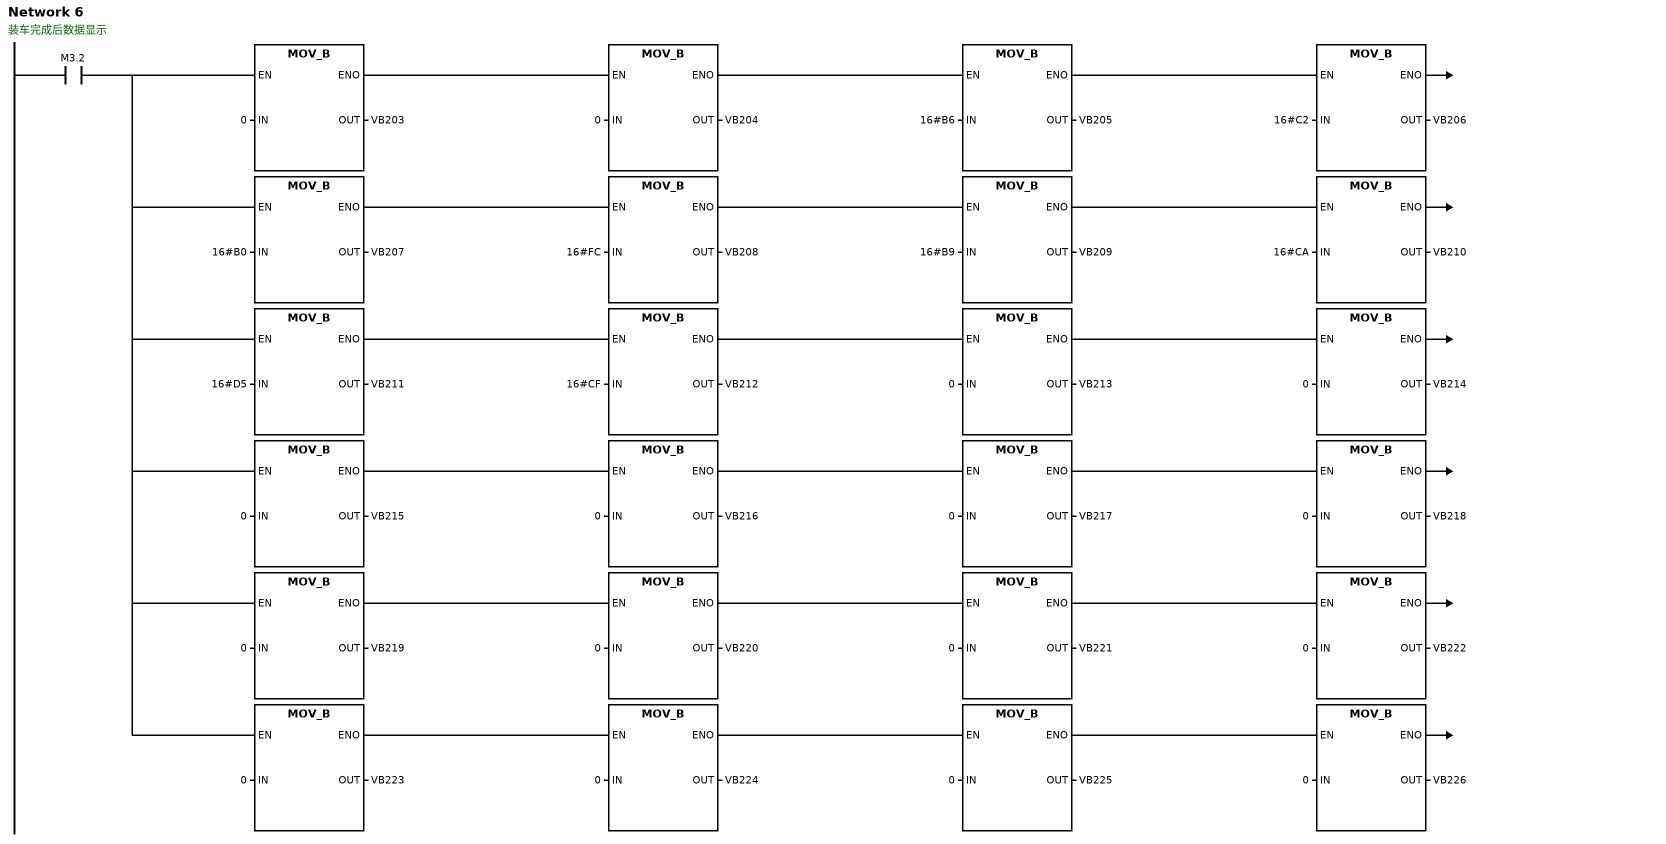
[picture p24: SBR12 networks 6-6]
Network 6
// 装车完成后数据显示
LD     M3.2
LPS
MOVB   0, VB203
AENO
MOVB   0, VB204
AENO
MOVB   16#B6, VB205
AENO
MOVB   16#C2, VB206
LRD
MOVB   16#B0, VB207
AENO
MOVB   16#FC, VB208
AENO
MOVB   16#B9, VB209
AENO
MOVB   16#CA, VB210
LRD
MOVB   16#D5, VB211
AENO
MOVB   16#CF, VB212
AENO
MOVB   0, VB213
AENO
MOVB   0, VB214
LRD
MOVB   0, VB215
AENO
MOVB   0, VB216
AENO
MOVB   0, VB217
AENO
MOVB   0, VB218
LRD
MOVB   0, VB219
AENO
MOVB   0, VB220
AENO
MOVB   0, VB221
AENO
MOVB   0, VB222
LPP
MOVB   0, VB223
AENO
MOVB   0, VB224
AENO
MOVB   0, VB225
AENO
MOVB   0, VB226
END_SUBROUTINE_BLOCK

SUBROUTINE_BLOCK LED3:SBR13
TITLE=
VAR_INPUT
D1:BYTE;	// LB0 
D2:BYTE;	// LB1 
D3:BYTE;	// LB2 
D4:BYTE;	// LB3 
P1:BYTE;	// LB4 
P2:BYTE;	// LB5 
P3:BYTE;	// LB6 
P4:BYTE;	// LB7 
P5:BYTE;	// LB8 
P6:BYTE;	// LB9 
P7:BYTE;	// LB10 
P8:BYTE;	// LB11 
RUN:WORD;	// LW12 
END_VAR
BEGIN
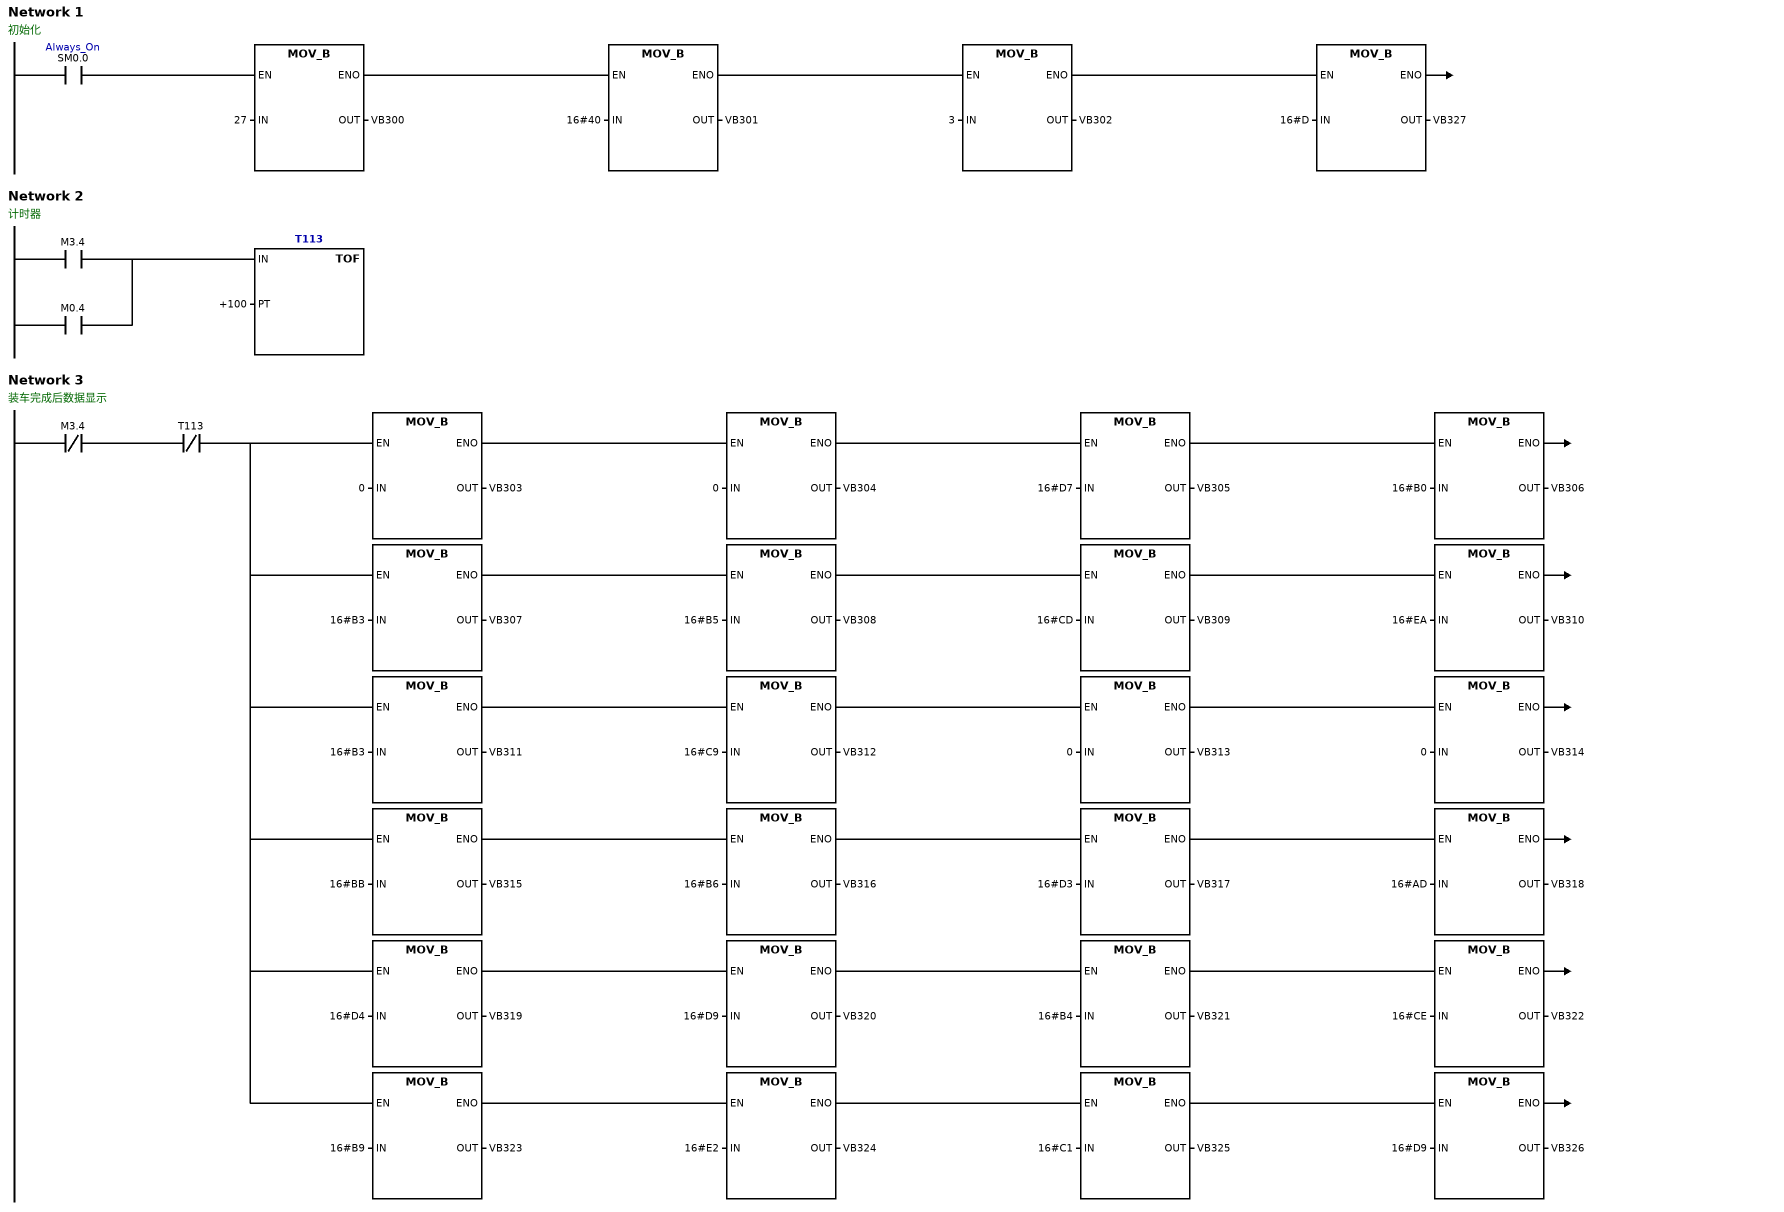
Network 1
// 初始化
LD     Always_On:SM0.0
MOVB   27, VB300
AENO
MOVB   16#40, VB301
AENO
MOVB   3, VB302
AENO
MOVB   16#D, VB327
Network 2
// 计时器
LD     M3.4
O      M0.4
TOF    T113, +100
Network 3
// 装车完成后数据显示
LDN    M3.4
AN     T113
LPS
MOVB   0, VB303
AENO
MOVB   0, VB304
AENO
MOVB   16#D7, VB305
AENO
MOVB   16#B0, VB306
LRD
MOVB   16#B3, VB307
AENO
MOVB   16#B5, VB308
AENO
MOVB   16#CD, VB309
AENO
MOVB   16#EA, VB310
LRD
MOVB   16#B3, VB311
AENO
MOVB   16#C9, VB312
AENO
MOVB   0, VB313
AENO
MOVB   0, VB314
LRD
MOVB   16#BB, VB315
AENO
MOVB   16#B6, VB316
AENO
MOVB   16#D3, VB317
AENO
MOVB   16#AD, VB318
LRD
MOVB   16#D4, VB319
AENO
MOVB   16#D9, VB320
AENO
MOVB   16#B4, VB321
AENO
MOVB   16#CE, VB322
LPP
MOVB   16#B9, VB323
AENO
MOVB   16#E2, VB324
AENO
MOVB   16#C1, VB325
AENO
MOVB   16#D9, VB326
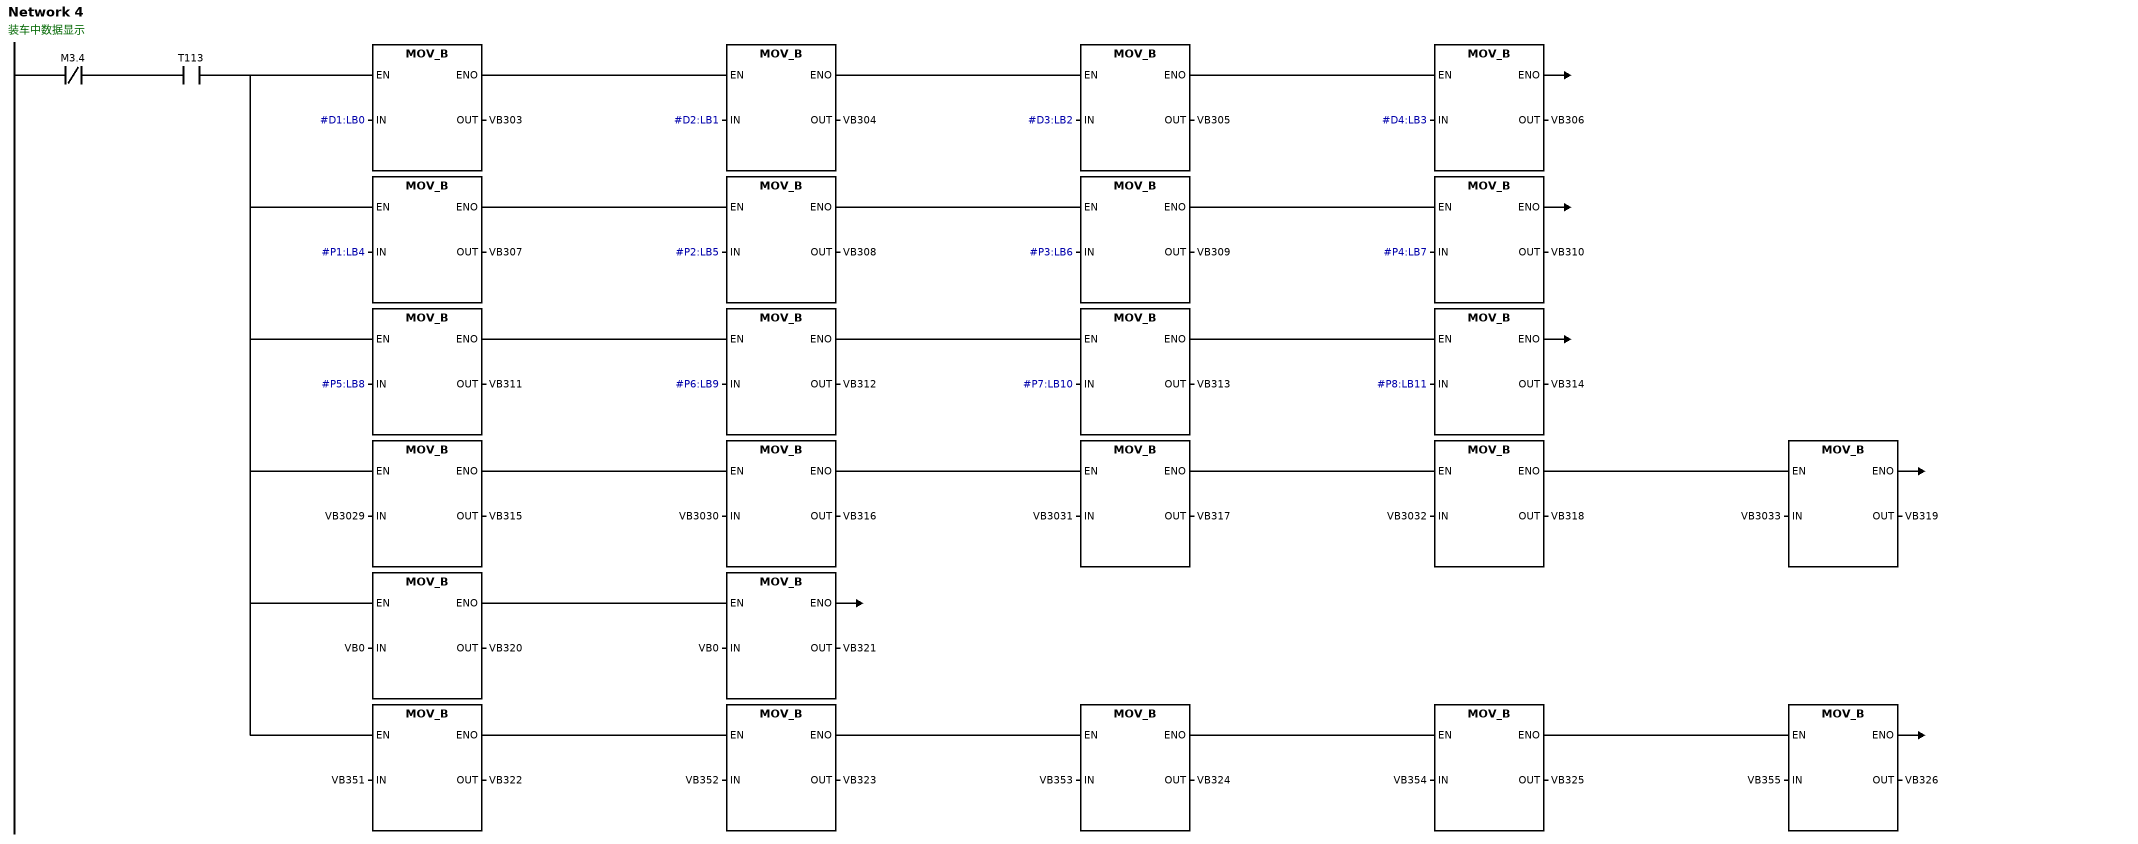
Network 4
// 装车中数据显示
LDN    M3.4
A      T113
LPS
MOVB   #D1:LB0, VB303
AENO
MOVB   #D2:LB1, VB304
AENO
MOVB   #D3:LB2, VB305
AENO
MOVB   #D4:LB3, VB306
LRD
MOVB   #P1:LB4, VB307
AENO
MOVB   #P2:LB5, VB308
AENO
MOVB   #P3:LB6, VB309
AENO
MOVB   #P4:LB7, VB310
LRD
MOVB   #P5:LB8, VB311
AENO
MOVB   #P6:LB9, VB312
AENO
MOVB   #P7:LB10, VB313
AENO
MOVB   #P8:LB11, VB314
LRD
MOVB   VB3029, VB315
AENO
MOVB   VB3030, VB316
AENO
MOVB   VB3031, VB317
AENO
MOVB   VB3032, VB318
AENO
MOVB   VB3033, VB319
LRD
MOVB   VB0, VB320
AENO
MOVB   VB0, VB321
LPP
MOVB   VB351, VB322
AENO
MOVB   VB352, VB323
AENO
MOVB   VB353, VB324
AENO
MOVB   VB354, VB325
AENO
MOVB   VB355, VB326
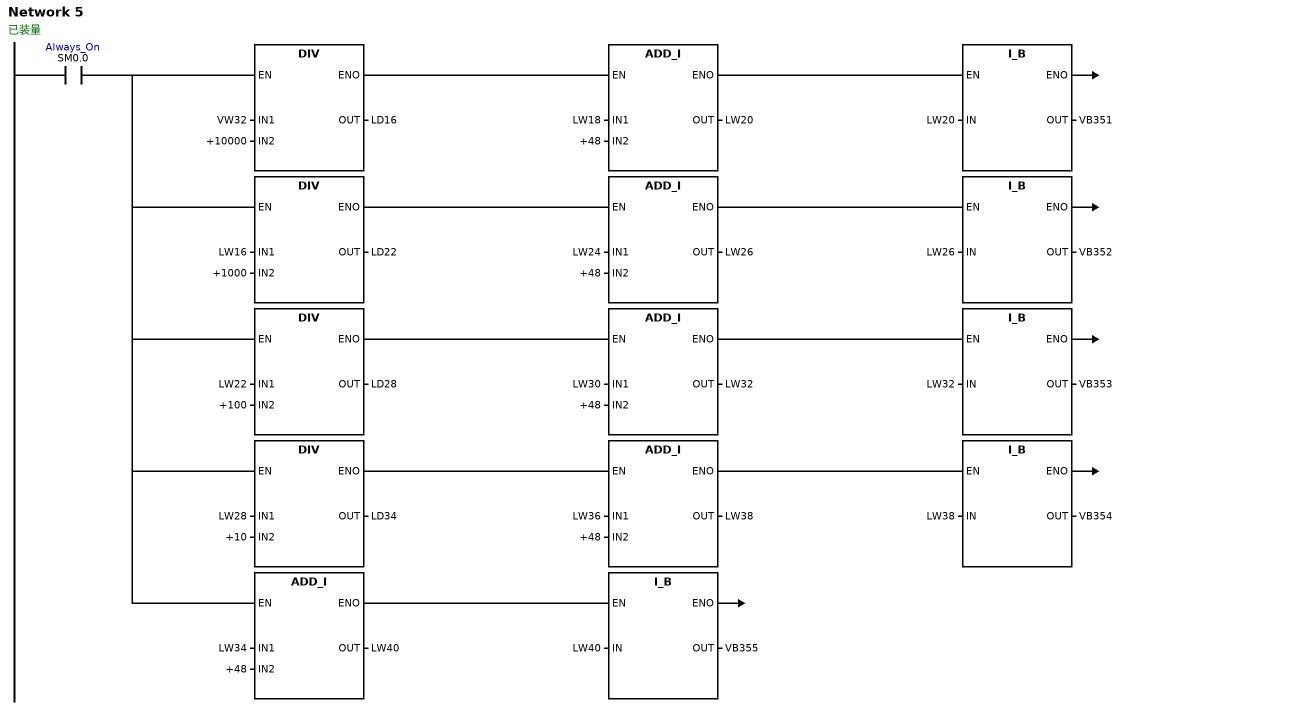
Network 5
// 已装量
LD     Always_On:SM0.0
LPS
MOVW   VW32, LW18
AENO
DIV    +10000, LD16
AENO
MOVW   LW18, LW20
AENO
+I     +48, LW20
AENO
ITB    LW20, VB351
LRD
MOVW   LW16, LW24
AENO
DIV    +1000, LD22
AENO
MOVW   LW24, LW26
AENO
+I     +48, LW26
AENO
ITB    LW26, VB352
LRD
MOVW   LW22, LW30
AENO
DIV    +100, LD28
AENO
MOVW   LW30, LW32
AENO
+I     +48, LW32
AENO
ITB    LW32, VB353
LRD
MOVW   LW28, LW36
AENO
DIV    +10, LD34
AENO
MOVW   LW36, LW38
AENO
+I     +48, LW38
AENO
ITB    LW38, VB354
LPP
MOVW   LW34, LW40
AENO
+I     +48, LW40
AENO
ITB    LW40, VB355
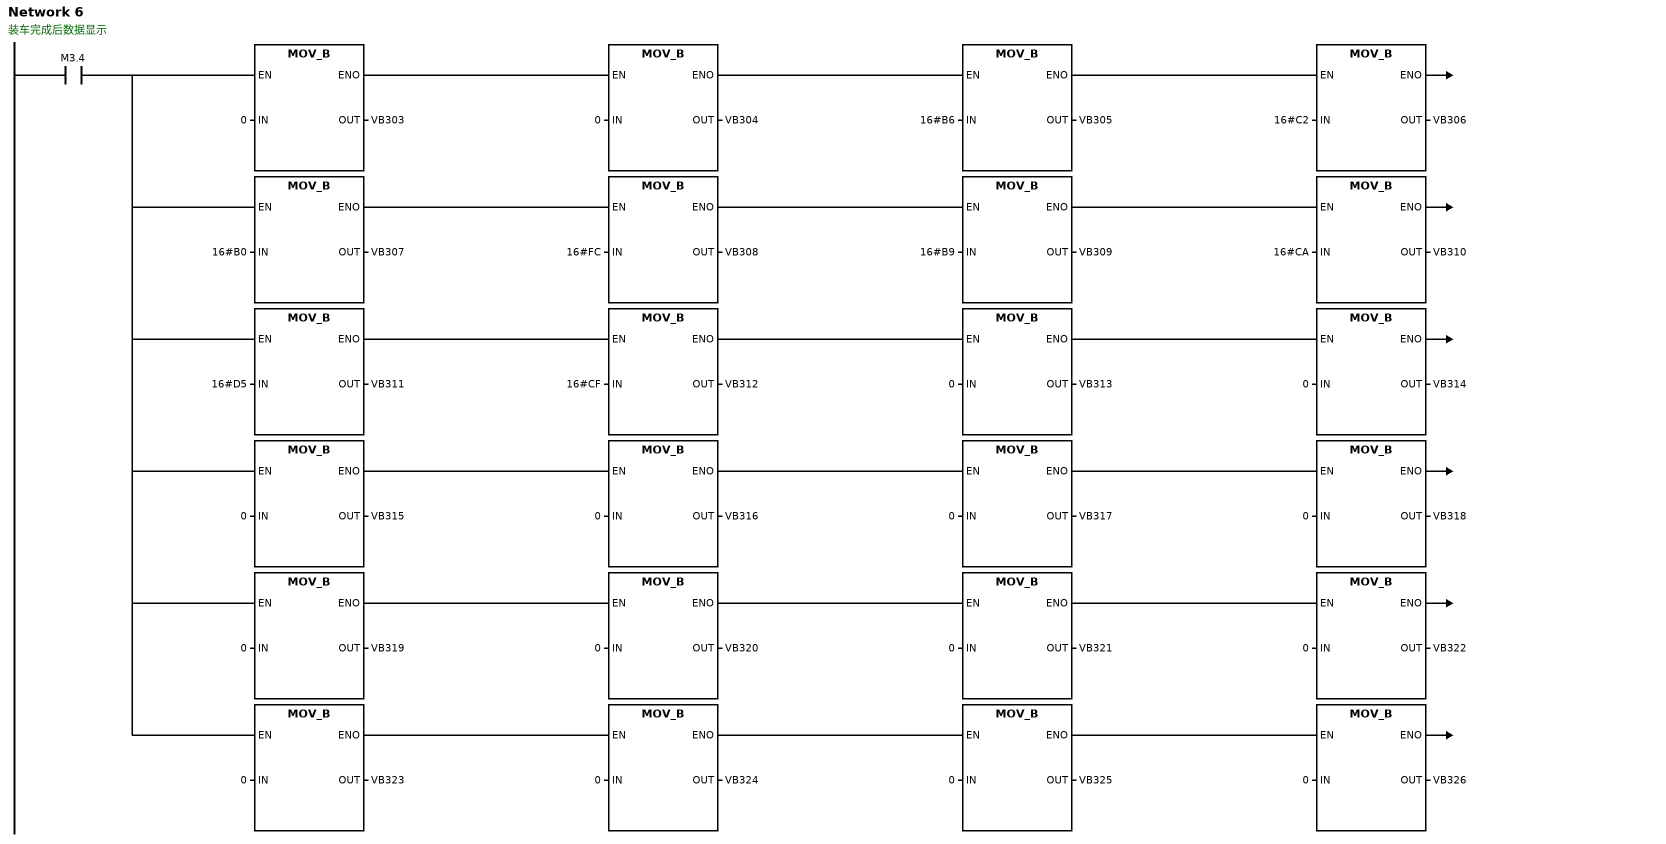
Network 6
// 装车完成后数据显示
LD     M3.4
LPS
MOVB   0, VB303
AENO
MOVB   0, VB304
AENO
MOVB   16#B6, VB305
AENO
MOVB   16#C2, VB306
LRD
MOVB   16#B0, VB307
AENO
MOVB   16#FC, VB308
AENO
MOVB   16#B9, VB309
AENO
MOVB   16#CA, VB310
LRD
MOVB   16#D5, VB311
AENO
MOVB   16#CF, VB312
AENO
MOVB   0, VB313
AENO
MOVB   0, VB314
LRD
MOVB   0, VB315
AENO
MOVB   0, VB316
AENO
MOVB   0, VB317
AENO
MOVB   0, VB318
LRD
MOVB   0, VB319
AENO
MOVB   0, VB320
AENO
MOVB   0, VB321
AENO
MOVB   0, VB322
LPP
MOVB   0, VB323
AENO
MOVB   0, VB324
AENO
MOVB   0, VB325
AENO
MOVB   0, VB326
END_SUBROUTINE_BLOCK

SUBROUTINE_BLOCK LED4:SBR14
TITLE=
VAR_INPUT
D1:BYTE;	// LB0 
D2:BYTE;	// LB1 
D3:BYTE;	// LB2 
D4:BYTE;	// LB3 
P1:BYTE;	// LB4 
P2:BYTE;	// LB5 
P3:BYTE;	// LB6 
P4:BYTE;	// LB7 
P5:BYTE;	// LB8 
P6:BYTE;	// LB9 
P7:BYTE;	// LB10 
P8:BYTE;	// LB11 
RUN:WORD;	// LW12 
END_VAR
BEGIN
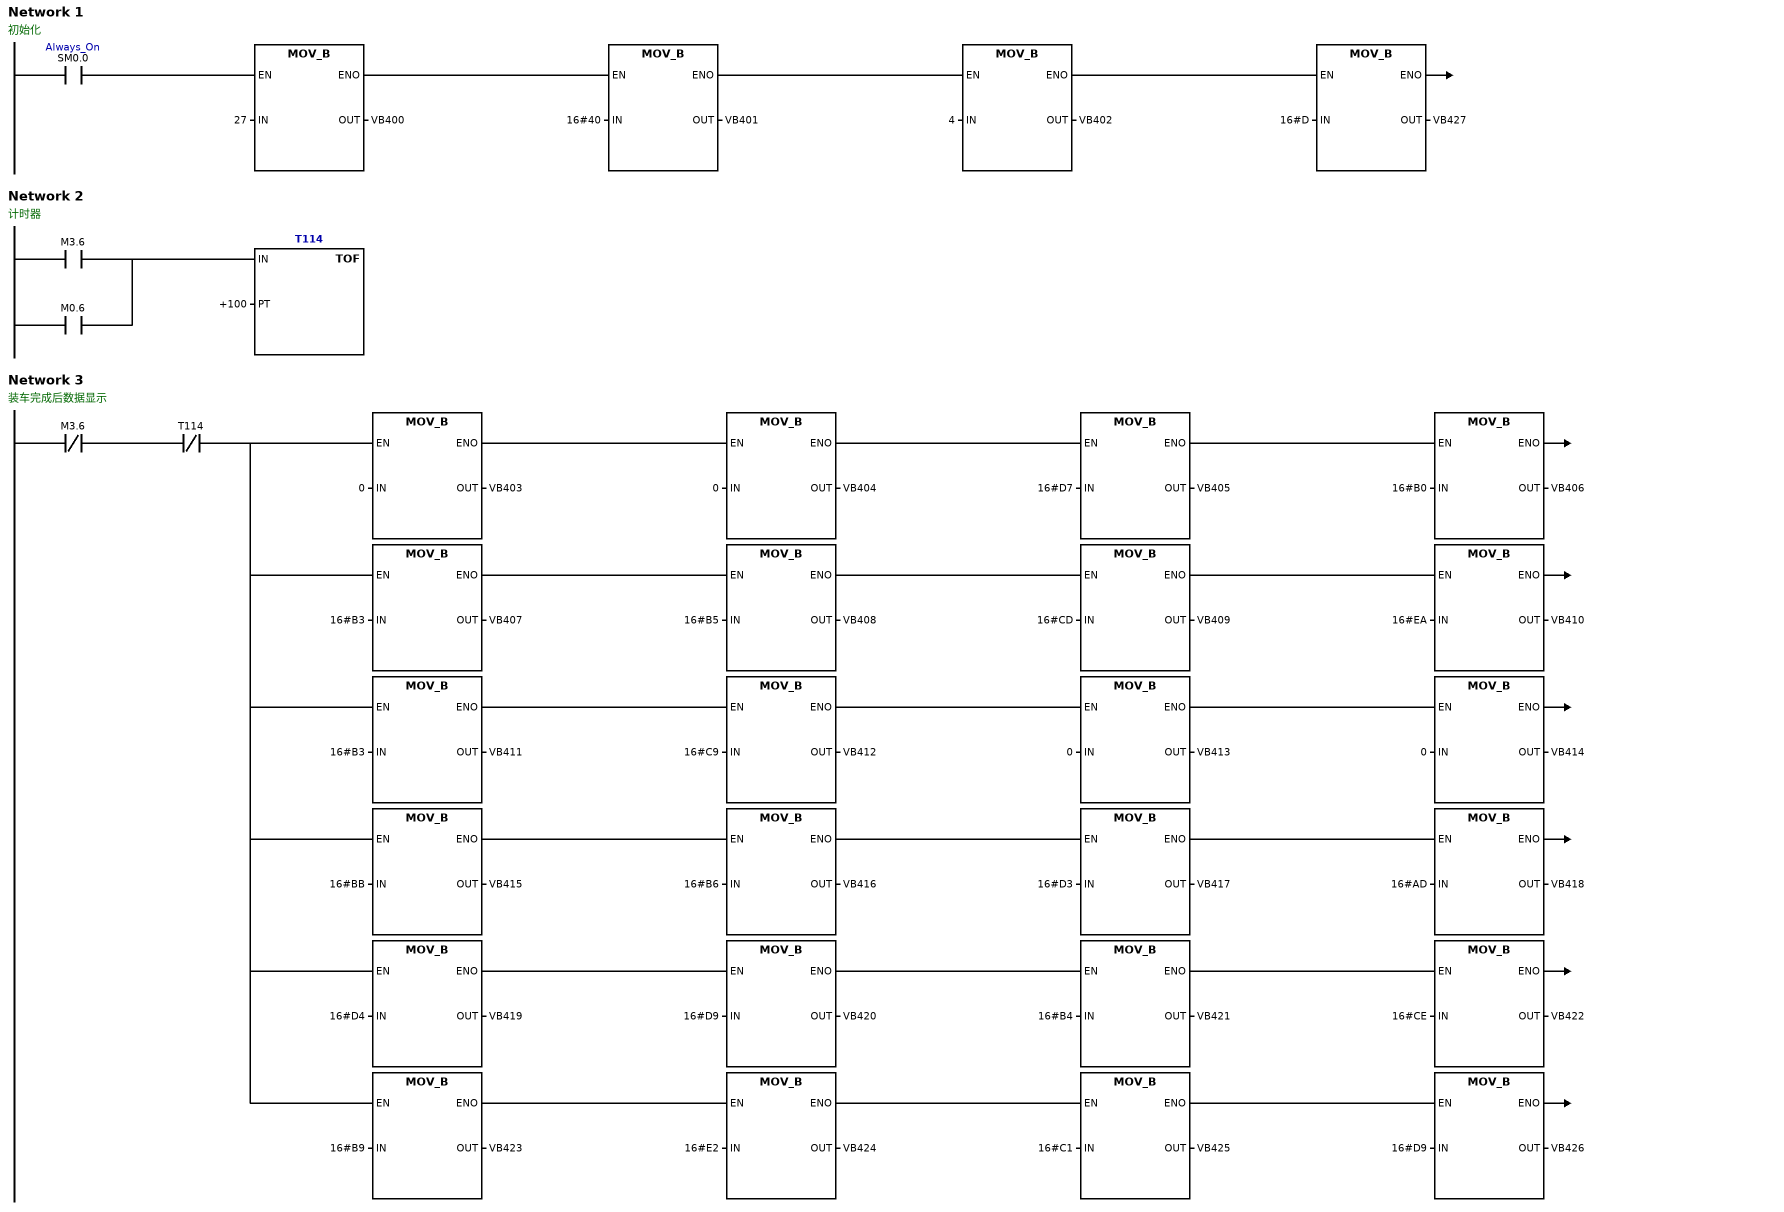
Network 1
// 初始化
LD     Always_On:SM0.0
MOVB   27, VB400
AENO
MOVB   16#40, VB401
AENO
MOVB   4, VB402
AENO
MOVB   16#D, VB427
Network 2
// 计时器
LD     M3.6
O      M0.6
TOF    T114, +100
Network 3
// 装车完成后数据显示
LDN    M3.6
AN     T114
LPS
MOVB   0, VB403
AENO
MOVB   0, VB404
AENO
MOVB   16#D7, VB405
AENO
MOVB   16#B0, VB406
LRD
MOVB   16#B3, VB407
AENO
MOVB   16#B5, VB408
AENO
MOVB   16#CD, VB409
AENO
MOVB   16#EA, VB410
LRD
MOVB   16#B3, VB411
AENO
MOVB   16#C9, VB412
AENO
MOVB   0, VB413
AENO
MOVB   0, VB414
LRD
MOVB   16#BB, VB415
AENO
MOVB   16#B6, VB416
AENO
MOVB   16#D3, VB417
AENO
MOVB   16#AD, VB418
LRD
MOVB   16#D4, VB419
AENO
MOVB   16#D9, VB420
AENO
MOVB   16#B4, VB421
AENO
MOVB   16#CE, VB422
LPP
MOVB   16#B9, VB423
AENO
MOVB   16#E2, VB424
AENO
MOVB   16#C1, VB425
AENO
MOVB   16#D9, VB426
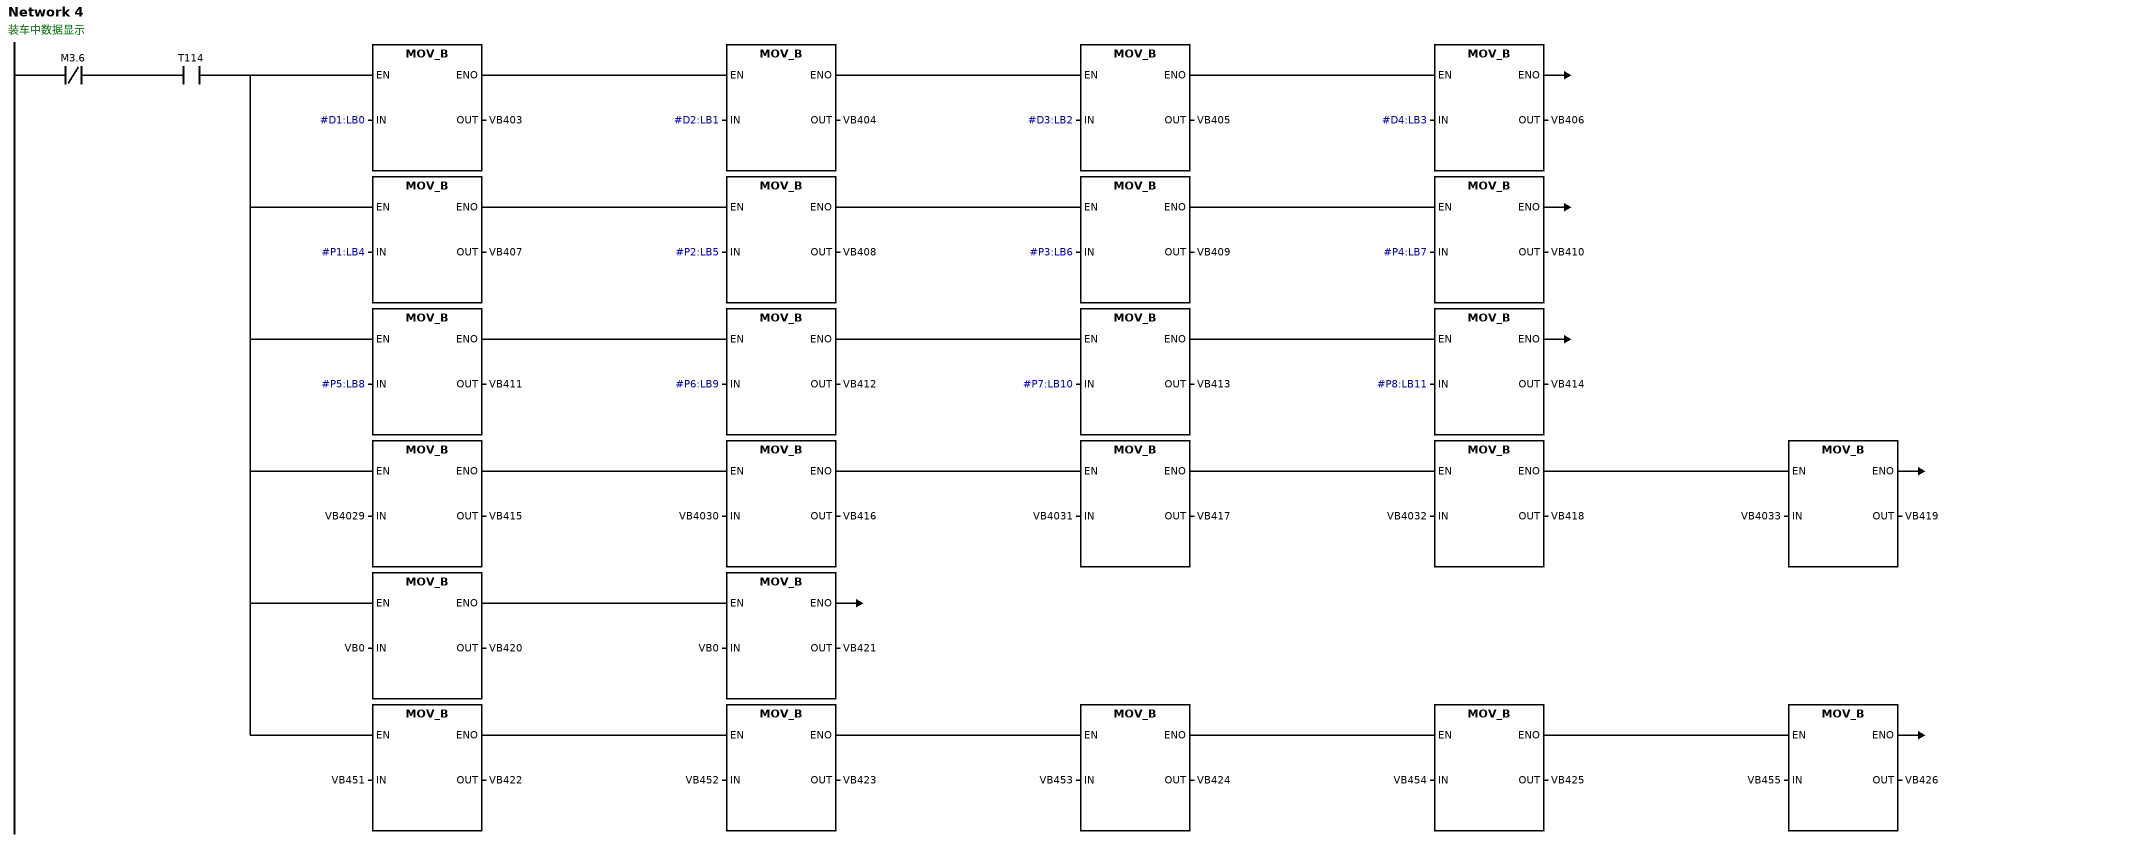
Network 4
// 装车中数据显示
LDN    M3.6
A      T114
LPS
MOVB   #D1:LB0, VB403
AENO
MOVB   #D2:LB1, VB404
AENO
MOVB   #D3:LB2, VB405
AENO
MOVB   #D4:LB3, VB406
LRD
MOVB   #P1:LB4, VB407
AENO
MOVB   #P2:LB5, VB408
AENO
MOVB   #P3:LB6, VB409
AENO
MOVB   #P4:LB7, VB410
LRD
MOVB   #P5:LB8, VB411
AENO
MOVB   #P6:LB9, VB412
AENO
MOVB   #P7:LB10, VB413
AENO
MOVB   #P8:LB11, VB414
LRD
MOVB   VB4029, VB415
AENO
MOVB   VB4030, VB416
AENO
MOVB   VB4031, VB417
AENO
MOVB   VB4032, VB418
AENO
MOVB   VB4033, VB419
LRD
MOVB   VB0, VB420
AENO
MOVB   VB0, VB421
LPP
MOVB   VB451, VB422
AENO
MOVB   VB452, VB423
AENO
MOVB   VB453, VB424
AENO
MOVB   VB454, VB425
AENO
MOVB   VB455, VB426
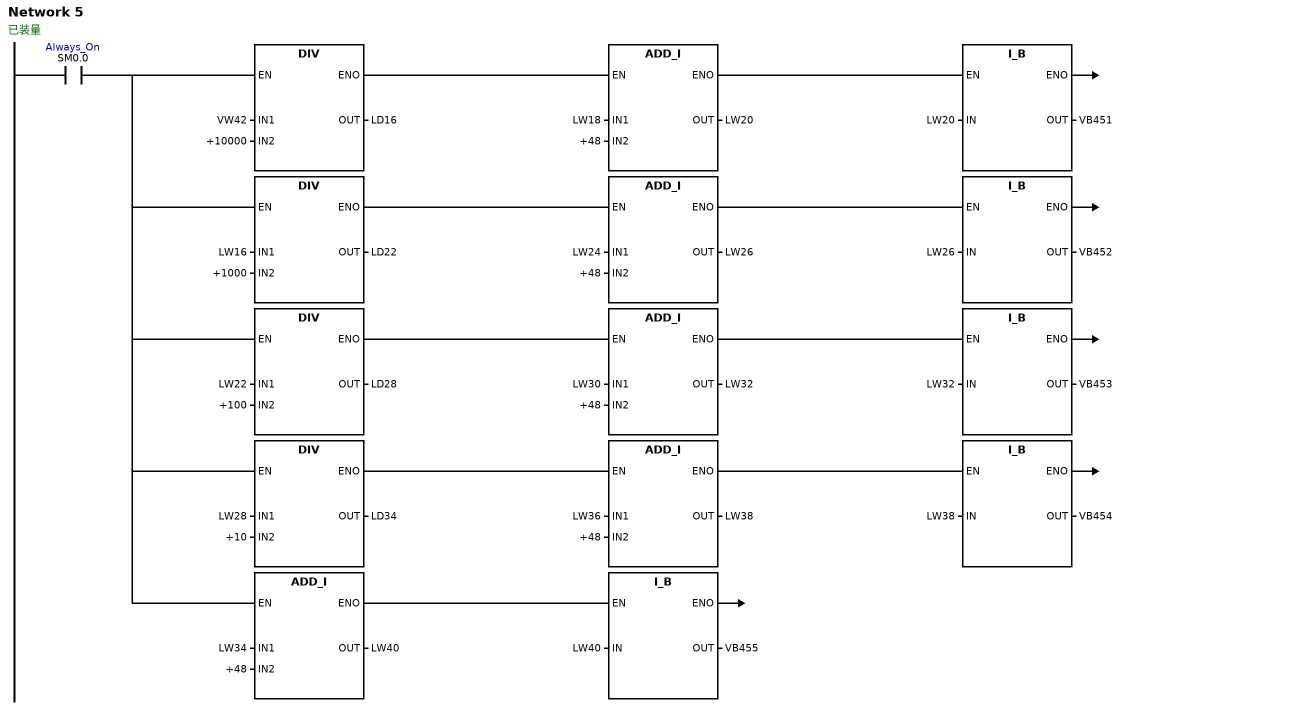
Network 5
// 已装量
LD     Always_On:SM0.0
LPS
MOVW   VW42, LW18
AENO
DIV    +10000, LD16
AENO
MOVW   LW18, LW20
AENO
+I     +48, LW20
AENO
ITB    LW20, VB451
LRD
MOVW   LW16, LW24
AENO
DIV    +1000, LD22
AENO
MOVW   LW24, LW26
AENO
+I     +48, LW26
AENO
ITB    LW26, VB452
LRD
MOVW   LW22, LW30
AENO
DIV    +100, LD28
AENO
MOVW   LW30, LW32
AENO
+I     +48, LW32
AENO
ITB    LW32, VB453
LRD
MOVW   LW28, LW36
AENO
DIV    +10, LD34
AENO
MOVW   LW36, LW38
AENO
+I     +48, LW38
AENO
ITB    LW38, VB454
LPP
MOVW   LW34, LW40
AENO
+I     +48, LW40
AENO
ITB    LW40, VB455
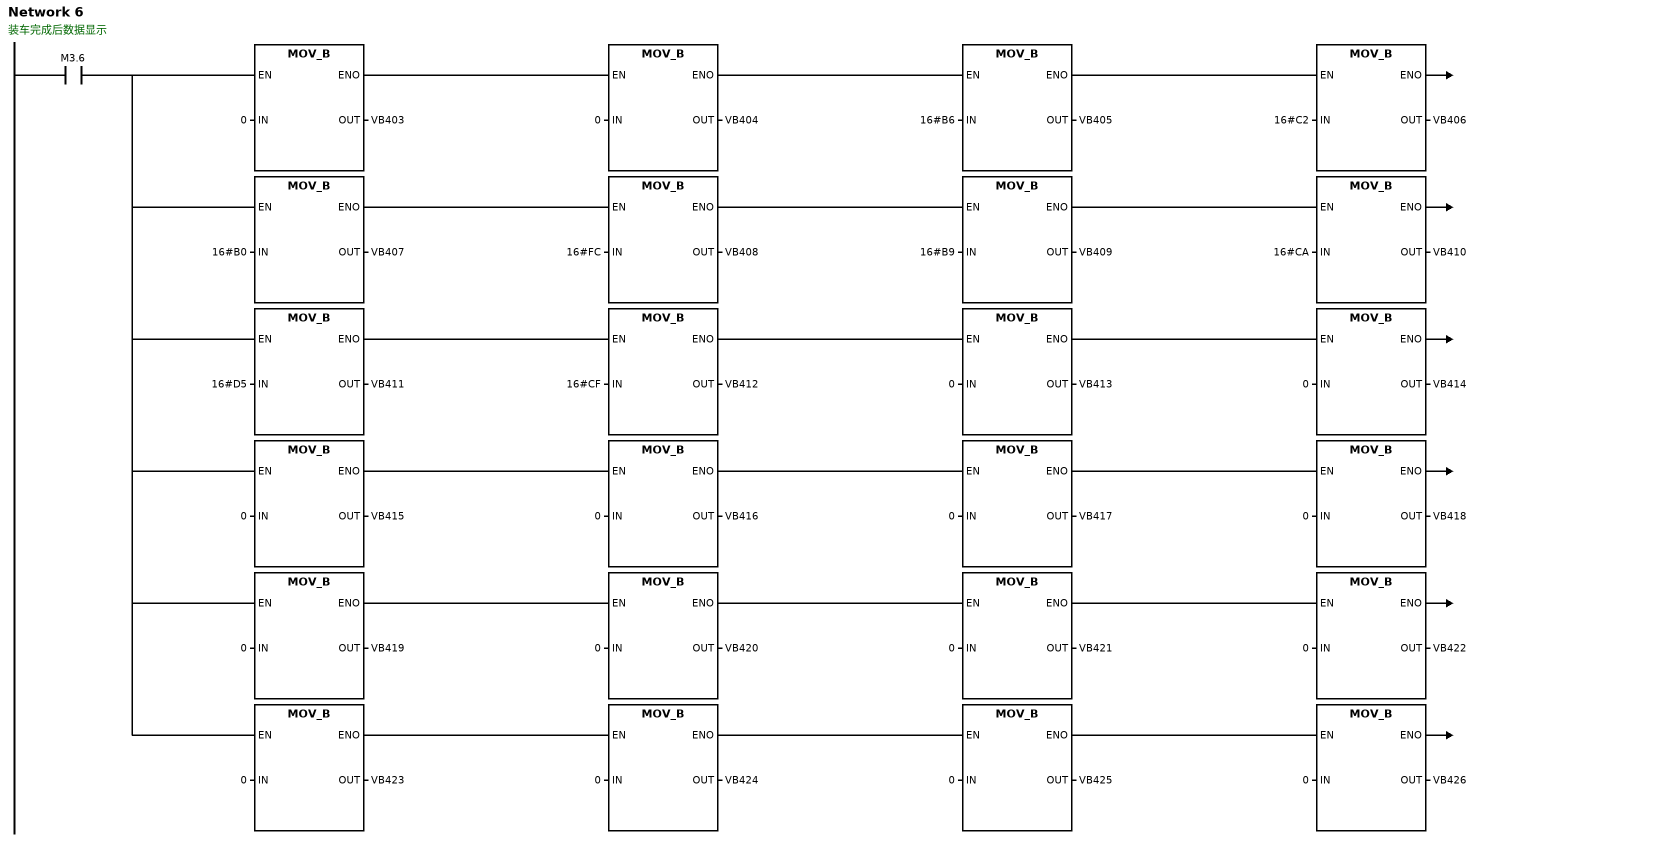
Network 6
// 装车完成后数据显示
LD     M3.6
LPS
MOVB   0, VB403
AENO
MOVB   0, VB404
AENO
MOVB   16#B6, VB405
AENO
MOVB   16#C2, VB406
LRD
MOVB   16#B0, VB407
AENO
MOVB   16#FC, VB408
AENO
MOVB   16#B9, VB409
AENO
MOVB   16#CA, VB410
LRD
MOVB   16#D5, VB411
AENO
MOVB   16#CF, VB412
AENO
MOVB   0, VB413
AENO
MOVB   0, VB414
LRD
MOVB   0, VB415
AENO
MOVB   0, VB416
AENO
MOVB   0, VB417
AENO
MOVB   0, VB418
LRD
MOVB   0, VB419
AENO
MOVB   0, VB420
AENO
MOVB   0, VB421
AENO
MOVB   0, VB422
LPP
MOVB   0, VB423
AENO
MOVB   0, VB424
AENO
MOVB   0, VB425
AENO
MOVB   0, VB426
END_SUBROUTINE_BLOCK

SUBROUTINE_BLOCK N1收:SBR21
TITLE=
VAR_OUTPUT
总袋数1:WORD;	// LW0 
袋长1:WORD;	// LW2 
END_VAR
VAR
TEMP1:WORD;	// LW4 
TEMP2:WORD;	// LW6 
TEMP3:WORD;	// LW8 
TEMP4:WORD;	// LW10 
TEMP5:WORD;	// LW12 
TEMP6:WORD;	// LW14 
TEMP7:WORD;	// LW16 
TEMP8:WORD;	// LW18 
TEMP9:WORD;	// LW20 
TEMP10:WORD;	// LW22 
TEMP11:WORD;	// LW24 
TEMP12:WORD;	// LW26 
TEMP13:WORD;	// LW28 
TEMP14:WORD;	// LW30 
TEMP15:WORD;	// LW32 
TEMP16:WORD;	// LW34 
TEMP17:WORD;	// LW36 
TEMP18:WORD;	// LW38 
TEMP19:WORD;	// LW40 
TEMP20:WORD;	// LW42 
TEMP21:WORD;	// LW44 
END_VAR
BEGIN
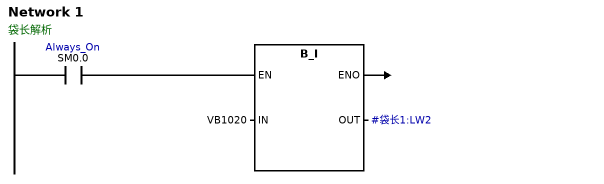
Network 1
// 袋长解析
LD     Always_On:SM0.0
BTI    VB1020, #袋长1:LW2
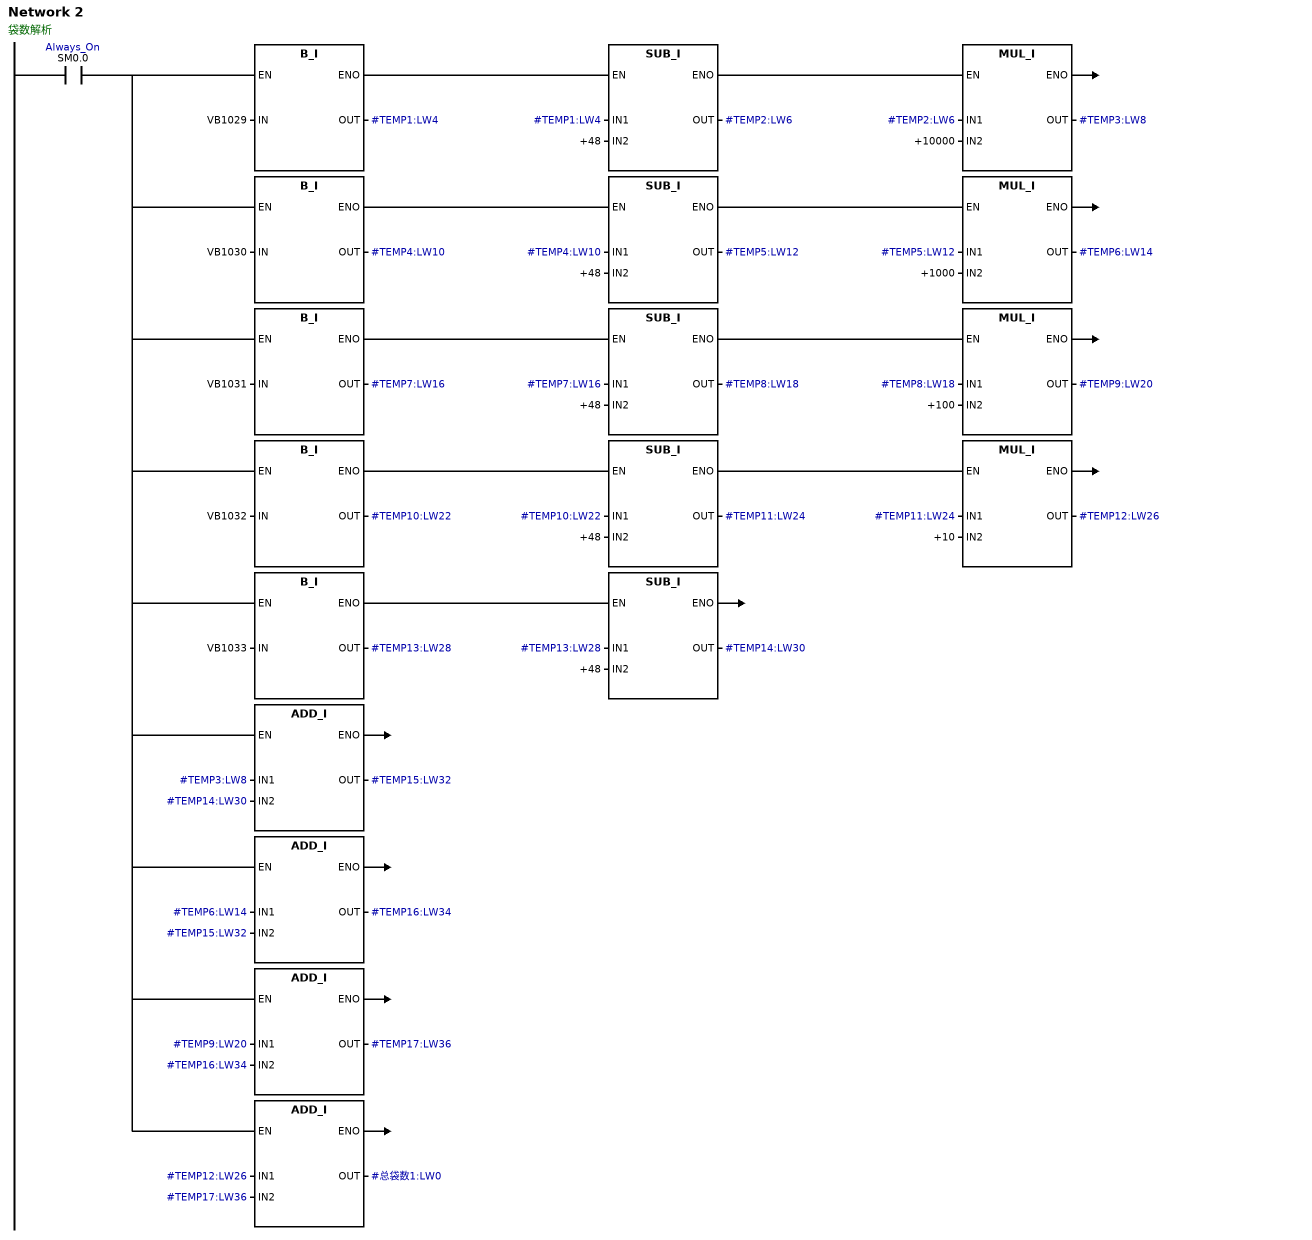
Network 2
// 袋数解析
LD     Always_On:SM0.0
LPS
BTI    VB1029, #TEMP1:LW4
AENO
MOVW   #TEMP1:LW4, #TEMP2:LW6
AENO
-I     +48, #TEMP2:LW6
AENO
MOVW   #TEMP2:LW6, #TEMP3:LW8
*I     +10000, #TEMP3:LW8
LRD
BTI    VB1030, #TEMP4:LW10
AENO
MOVW   #TEMP4:LW10, #TEMP5:LW12
AENO
-I     +48, #TEMP5:LW12
AENO
MOVW   #TEMP5:LW12, #TEMP6:LW14
*I     +1000, #TEMP6:LW14
LRD
BTI    VB1031, #TEMP7:LW16
AENO
MOVW   #TEMP7:LW16, #TEMP8:LW18
AENO
-I     +48, #TEMP8:LW18
AENO
MOVW   #TEMP8:LW18, #TEMP9:LW20
*I     +100, #TEMP9:LW20
LRD
BTI    VB1032, #TEMP10:LW22
AENO
MOVW   #TEMP10:LW22, #TEMP11:LW24
AENO
-I     +48, #TEMP11:LW24
AENO
MOVW   #TEMP11:LW24, #TEMP12:LW26
*I     +10, #TEMP12:LW26
LRD
BTI    VB1033, #TEMP13:LW28
AENO
MOVW   #TEMP13:LW28, #TEMP14:LW30
-I     +48, #TEMP14:LW30
LRD
MOVW   #TEMP3:LW8, #TEMP15:LW32
+I     #TEMP14:LW30, #TEMP15:LW32
LRD
MOVW   #TEMP6:LW14, #TEMP16:LW34
+I     #TEMP15:LW32, #TEMP16:LW34
LRD
MOVW   #TEMP9:LW20, #TEMP17:LW36
+I     #TEMP16:LW34, #TEMP17:LW36
LPP
MOVW   #TEMP12:LW26, #总袋数1:LW0
+I     #TEMP17:LW36, #总袋数1:LW0
END_SUBROUTINE_BLOCK

SUBROUTINE_BLOCK N2收:SBR22
TITLE=
VAR_OUTPUT
总袋数1:WORD;	// LW0 
袋长1:WORD;	// LW2 
END_VAR
VAR
TEMP1:WORD;	// LW4 
TEMP2:WORD;	// LW6 
TEMP3:WORD;	// LW8 
TEMP4:WORD;	// LW10 
TEMP5:WORD;	// LW12 
TEMP6:WORD;	// LW14 
TEMP7:WORD;	// LW16 
TEMP8:WORD;	// LW18 
TEMP9:WORD;	// LW20 
TEMP10:WORD;	// LW22 
TEMP11:WORD;	// LW24 
TEMP12:WORD;	// LW26 
TEMP13:WORD;	// LW28 
TEMP14:WORD;	// LW30 
TEMP15:WORD;	// LW32 
TEMP16:WORD;	// LW34 
TEMP17:WORD;	// LW36 
TEMP18:WORD;	// LW38 
TEMP19:WORD;	// LW40 
TEMP20:WORD;	// LW42 
TEMP21:WORD;	// LW44 
END_VAR
BEGIN
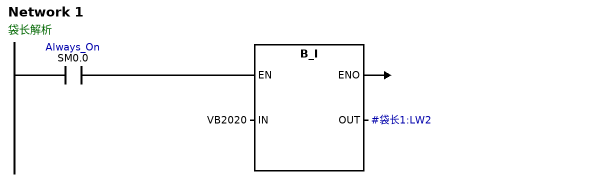
Network 1
// 袋长解析
LD     Always_On:SM0.0
BTI    VB2020, #袋长1:LW2
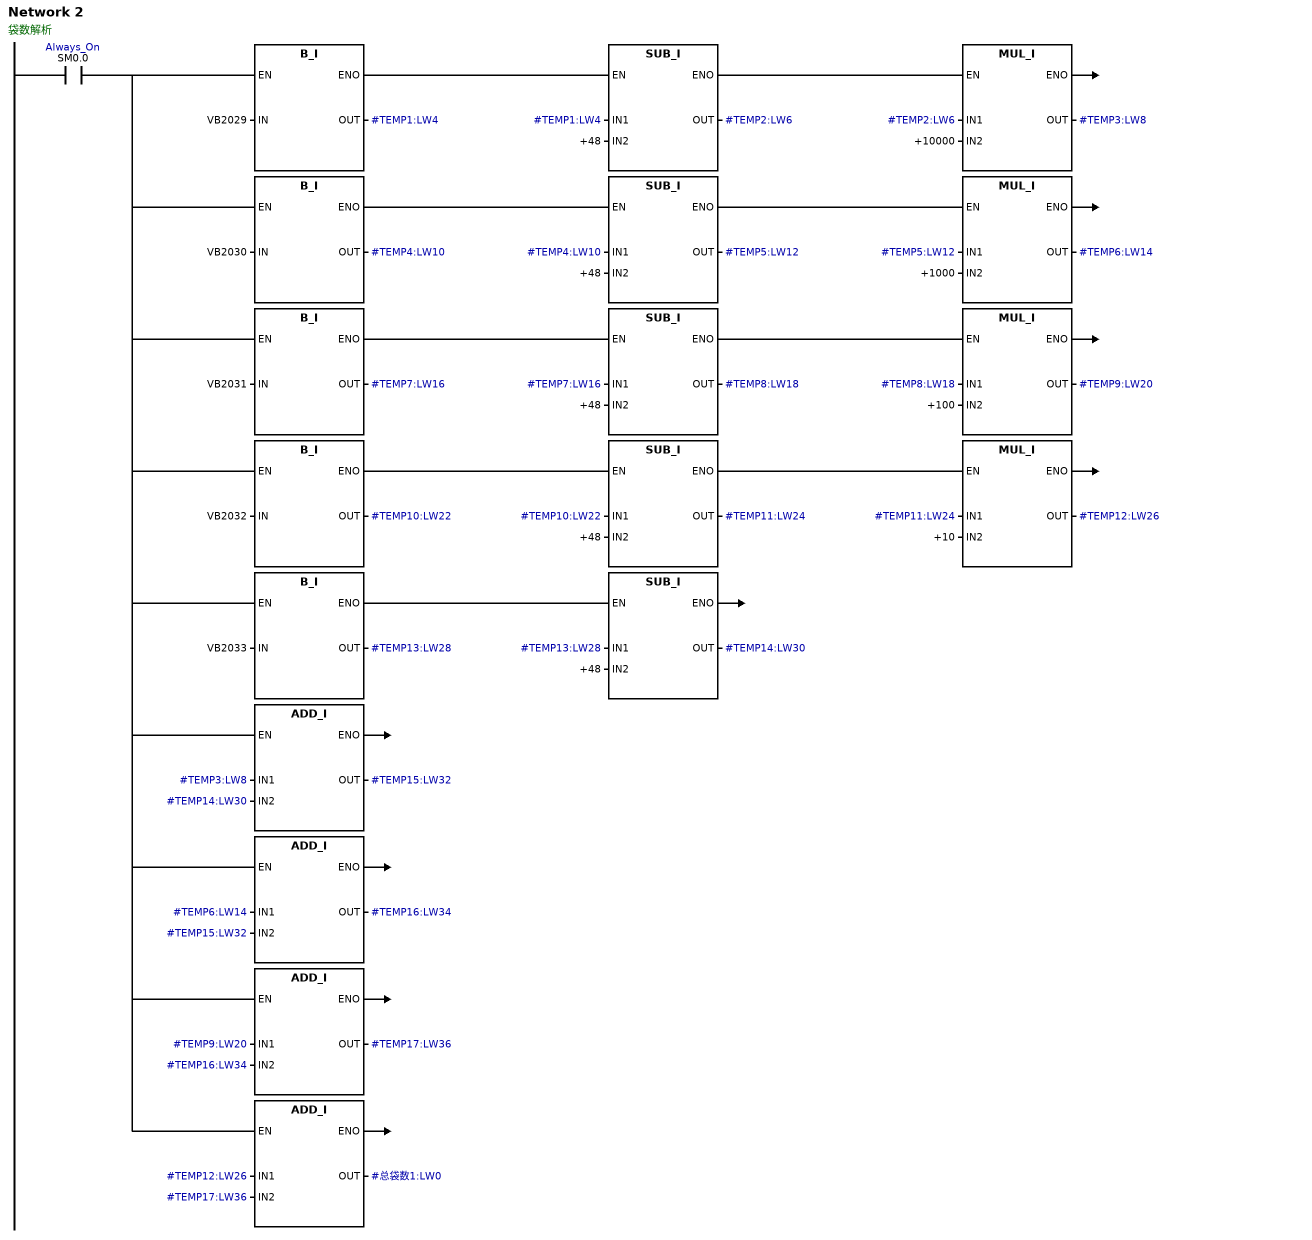
Network 2
// 袋数解析
LD     Always_On:SM0.0
LPS
BTI    VB2029, #TEMP1:LW4
AENO
MOVW   #TEMP1:LW4, #TEMP2:LW6
AENO
-I     +48, #TEMP2:LW6
AENO
MOVW   #TEMP2:LW6, #TEMP3:LW8
*I     +10000, #TEMP3:LW8
LRD
BTI    VB2030, #TEMP4:LW10
AENO
MOVW   #TEMP4:LW10, #TEMP5:LW12
AENO
-I     +48, #TEMP5:LW12
AENO
MOVW   #TEMP5:LW12, #TEMP6:LW14
*I     +1000, #TEMP6:LW14
LRD
BTI    VB2031, #TEMP7:LW16
AENO
MOVW   #TEMP7:LW16, #TEMP8:LW18
AENO
-I     +48, #TEMP8:LW18
AENO
MOVW   #TEMP8:LW18, #TEMP9:LW20
*I     +100, #TEMP9:LW20
LRD
BTI    VB2032, #TEMP10:LW22
AENO
MOVW   #TEMP10:LW22, #TEMP11:LW24
AENO
-I     +48, #TEMP11:LW24
AENO
MOVW   #TEMP11:LW24, #TEMP12:LW26
*I     +10, #TEMP12:LW26
LRD
BTI    VB2033, #TEMP13:LW28
AENO
MOVW   #TEMP13:LW28, #TEMP14:LW30
-I     +48, #TEMP14:LW30
LRD
MOVW   #TEMP3:LW8, #TEMP15:LW32
+I     #TEMP14:LW30, #TEMP15:LW32
LRD
MOVW   #TEMP6:LW14, #TEMP16:LW34
+I     #TEMP15:LW32, #TEMP16:LW34
LRD
MOVW   #TEMP9:LW20, #TEMP17:LW36
+I     #TEMP16:LW34, #TEMP17:LW36
LPP
MOVW   #TEMP12:LW26, #总袋数1:LW0
+I     #TEMP17:LW36, #总袋数1:LW0
END_SUBROUTINE_BLOCK

SUBROUTINE_BLOCK N3收:SBR23
TITLE=
VAR_OUTPUT
总袋数1:WORD;	// LW0 
袋长1:WORD;	// LW2 
END_VAR
VAR
TEMP1:WORD;	// LW4 
TEMP2:WORD;	// LW6 
TEMP3:WORD;	// LW8 
TEMP4:WORD;	// LW10 
TEMP5:WORD;	// LW12 
TEMP6:WORD;	// LW14 
TEMP7:WORD;	// LW16 
TEMP8:WORD;	// LW18 
TEMP9:WORD;	// LW20 
TEMP10:WORD;	// LW22 
TEMP11:WORD;	// LW24 
TEMP12:WORD;	// LW26 
TEMP13:WORD;	// LW28 
TEMP14:WORD;	// LW30 
TEMP15:WORD;	// LW32 
TEMP16:WORD;	// LW34 
TEMP17:WORD;	// LW36 
TEMP18:WORD;	// LW38 
TEMP19:WORD;	// LW40 
TEMP20:WORD;	// LW42 
TEMP21:WORD;	// LW44 
END_VAR
BEGIN
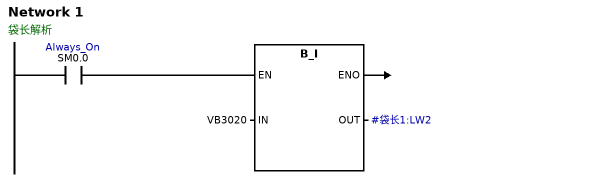
Network 1
// 袋长解析
LD     Always_On:SM0.0
BTI    VB3020, #袋长1:LW2
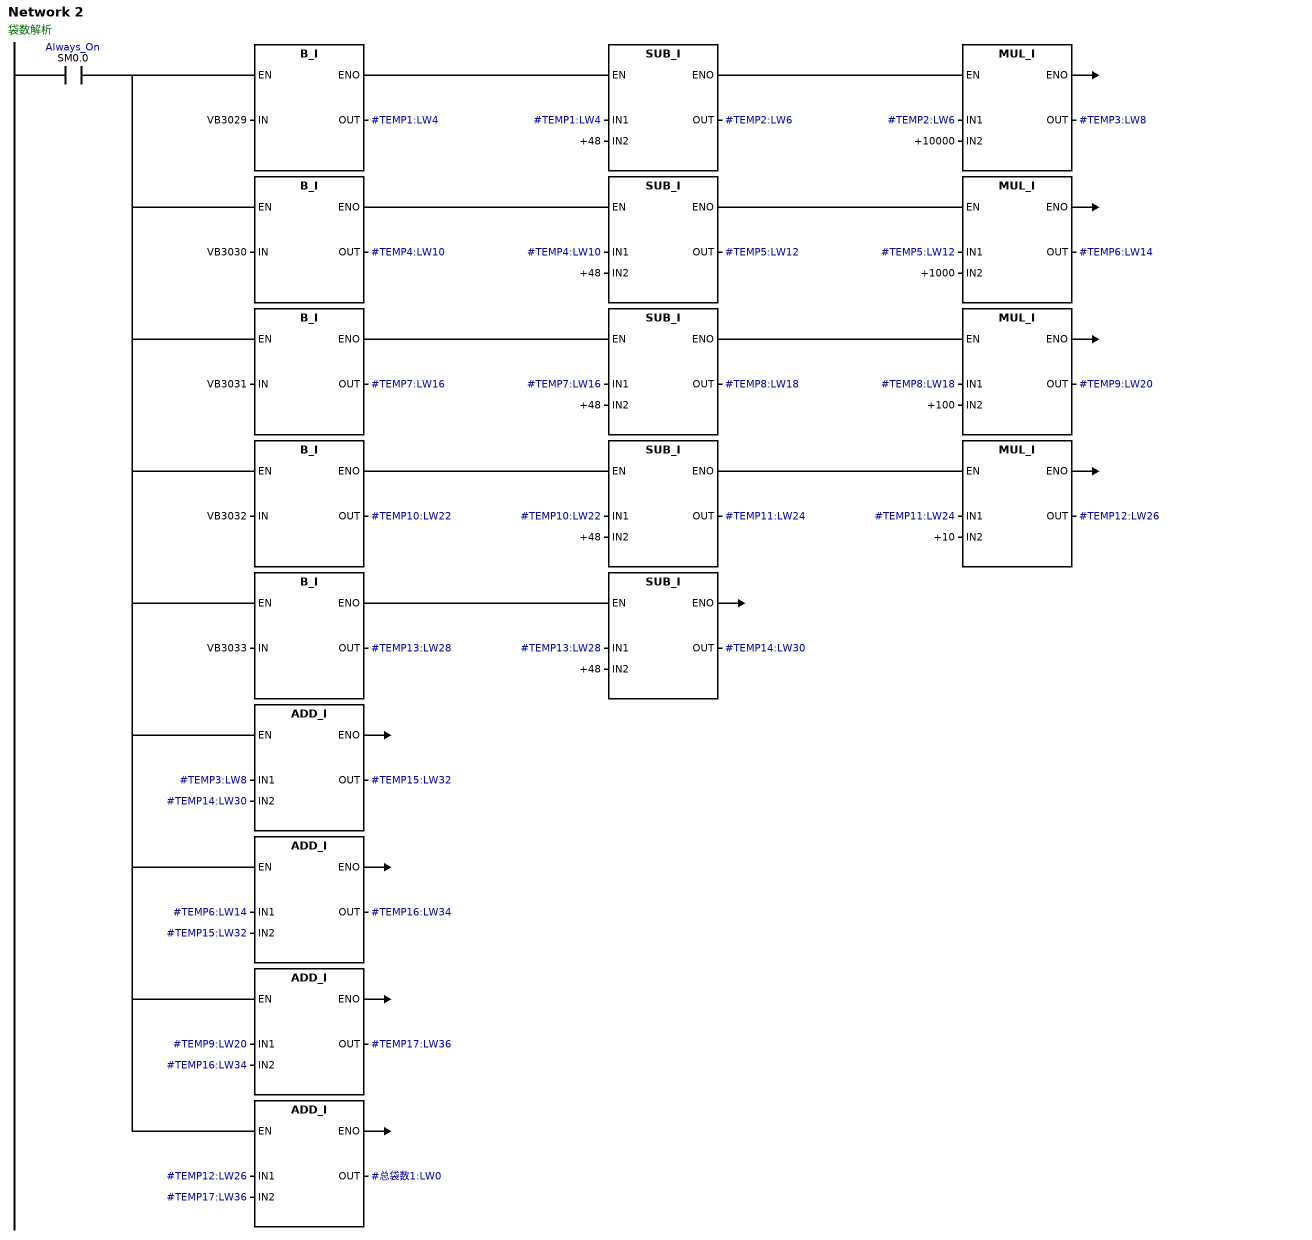
Network 2
// 袋数解析
LD     Always_On:SM0.0
LPS
BTI    VB3029, #TEMP1:LW4
AENO
MOVW   #TEMP1:LW4, #TEMP2:LW6
AENO
-I     +48, #TEMP2:LW6
AENO
MOVW   #TEMP2:LW6, #TEMP3:LW8
*I     +10000, #TEMP3:LW8
LRD
BTI    VB3030, #TEMP4:LW10
AENO
MOVW   #TEMP4:LW10, #TEMP5:LW12
AENO
-I     +48, #TEMP5:LW12
AENO
MOVW   #TEMP5:LW12, #TEMP6:LW14
*I     +1000, #TEMP6:LW14
LRD
BTI    VB3031, #TEMP7:LW16
AENO
MOVW   #TEMP7:LW16, #TEMP8:LW18
AENO
-I     +48, #TEMP8:LW18
AENO
MOVW   #TEMP8:LW18, #TEMP9:LW20
*I     +100, #TEMP9:LW20
LRD
BTI    VB3032, #TEMP10:LW22
AENO
MOVW   #TEMP10:LW22, #TEMP11:LW24
AENO
-I     +48, #TEMP11:LW24
AENO
MOVW   #TEMP11:LW24, #TEMP12:LW26
*I     +10, #TEMP12:LW26
LRD
BTI    VB3033, #TEMP13:LW28
AENO
MOVW   #TEMP13:LW28, #TEMP14:LW30
-I     +48, #TEMP14:LW30
LRD
MOVW   #TEMP3:LW8, #TEMP15:LW32
+I     #TEMP14:LW30, #TEMP15:LW32
LRD
MOVW   #TEMP6:LW14, #TEMP16:LW34
+I     #TEMP15:LW32, #TEMP16:LW34
LRD
MOVW   #TEMP9:LW20, #TEMP17:LW36
+I     #TEMP16:LW34, #TEMP17:LW36
LPP
MOVW   #TEMP12:LW26, #总袋数1:LW0
+I     #TEMP17:LW36, #总袋数1:LW0
END_SUBROUTINE_BLOCK

SUBROUTINE_BLOCK N4收:SBR24
TITLE=
VAR_OUTPUT
总袋数1:WORD;	// LW0 
袋长1:WORD;	// LW2 
END_VAR
VAR
TEMP1:WORD;	// LW4 
TEMP2:WORD;	// LW6 
TEMP3:WORD;	// LW8 
TEMP4:WORD;	// LW10 
TEMP5:WORD;	// LW12 
TEMP6:WORD;	// LW14 
TEMP7:WORD;	// LW16 
TEMP8:WORD;	// LW18 
TEMP9:WORD;	// LW20 
TEMP10:WORD;	// LW22 
TEMP11:WORD;	// LW24 
TEMP12:WORD;	// LW26 
TEMP13:WORD;	// LW28 
TEMP14:WORD;	// LW30 
TEMP15:WORD;	// LW32 
TEMP16:WORD;	// LW34 
TEMP17:WORD;	// LW36 
TEMP18:WORD;	// LW38 
TEMP19:WORD;	// LW40 
TEMP20:WORD;	// LW42 
TEMP21:WORD;	// LW44 
END_VAR
BEGIN
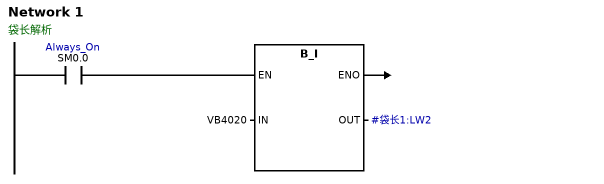
Network 1
// 袋长解析
LD     Always_On:SM0.0
BTI    VB4020, #袋长1:LW2
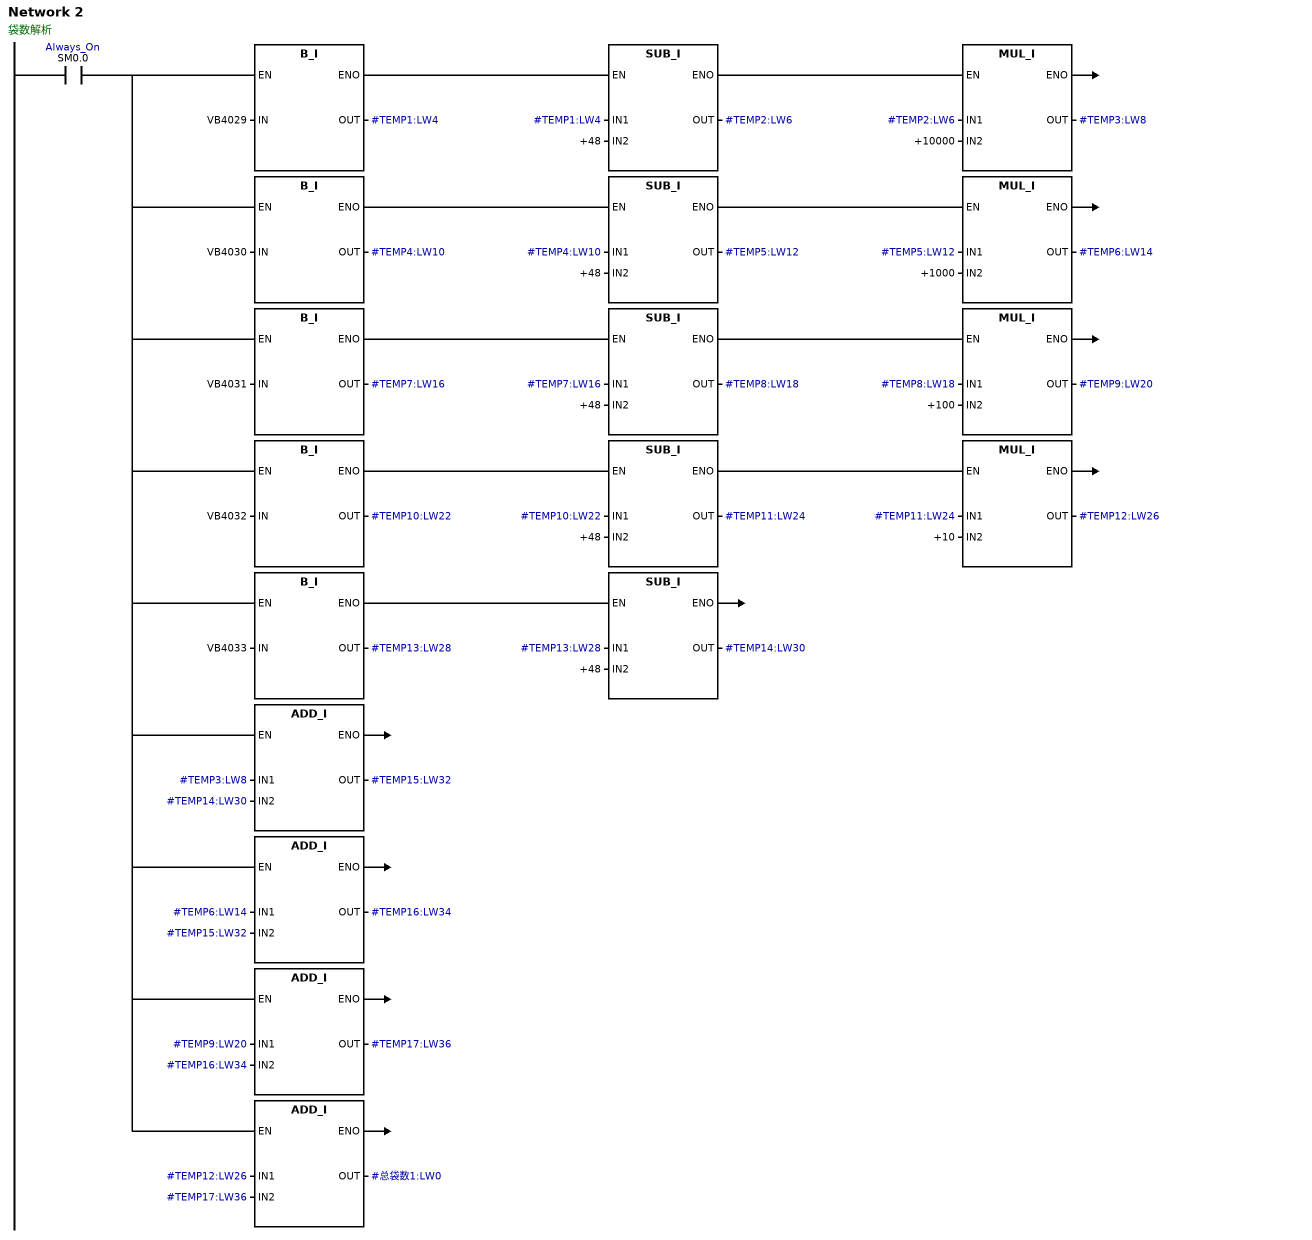
Network 2
// 袋数解析
LD     Always_On:SM0.0
LPS
BTI    VB4029, #TEMP1:LW4
AENO
MOVW   #TEMP1:LW4, #TEMP2:LW6
AENO
-I     +48, #TEMP2:LW6
AENO
MOVW   #TEMP2:LW6, #TEMP3:LW8
*I     +10000, #TEMP3:LW8
LRD
BTI    VB4030, #TEMP4:LW10
AENO
MOVW   #TEMP4:LW10, #TEMP5:LW12
AENO
-I     +48, #TEMP5:LW12
AENO
MOVW   #TEMP5:LW12, #TEMP6:LW14
*I     +1000, #TEMP6:LW14
LRD
BTI    VB4031, #TEMP7:LW16
AENO
MOVW   #TEMP7:LW16, #TEMP8:LW18
AENO
-I     +48, #TEMP8:LW18
AENO
MOVW   #TEMP8:LW18, #TEMP9:LW20
*I     +100, #TEMP9:LW20
LRD
BTI    VB4032, #TEMP10:LW22
AENO
MOVW   #TEMP10:LW22, #TEMP11:LW24
AENO
-I     +48, #TEMP11:LW24
AENO
MOVW   #TEMP11:LW24, #TEMP12:LW26
*I     +10, #TEMP12:LW26
LRD
BTI    VB4033, #TEMP13:LW28
AENO
MOVW   #TEMP13:LW28, #TEMP14:LW30
-I     +48, #TEMP14:LW30
LRD
MOVW   #TEMP3:LW8, #TEMP15:LW32
+I     #TEMP14:LW30, #TEMP15:LW32
LRD
MOVW   #TEMP6:LW14, #TEMP16:LW34
+I     #TEMP15:LW32, #TEMP16:LW34
LRD
MOVW   #TEMP9:LW20, #TEMP17:LW36
+I     #TEMP16:LW34, #TEMP17:LW36
LPP
MOVW   #TEMP12:LW26, #总袋数1:LW0
+I     #TEMP17:LW36, #总袋数1:LW0
END_SUBROUTINE_BLOCK

SUBROUTINE_BLOCK GGLED1_2:SBR31
TITLE=子程序注释
VAR_INPUT
屏3地址:BYTE;	// LB0 
END_VAR
BEGIN
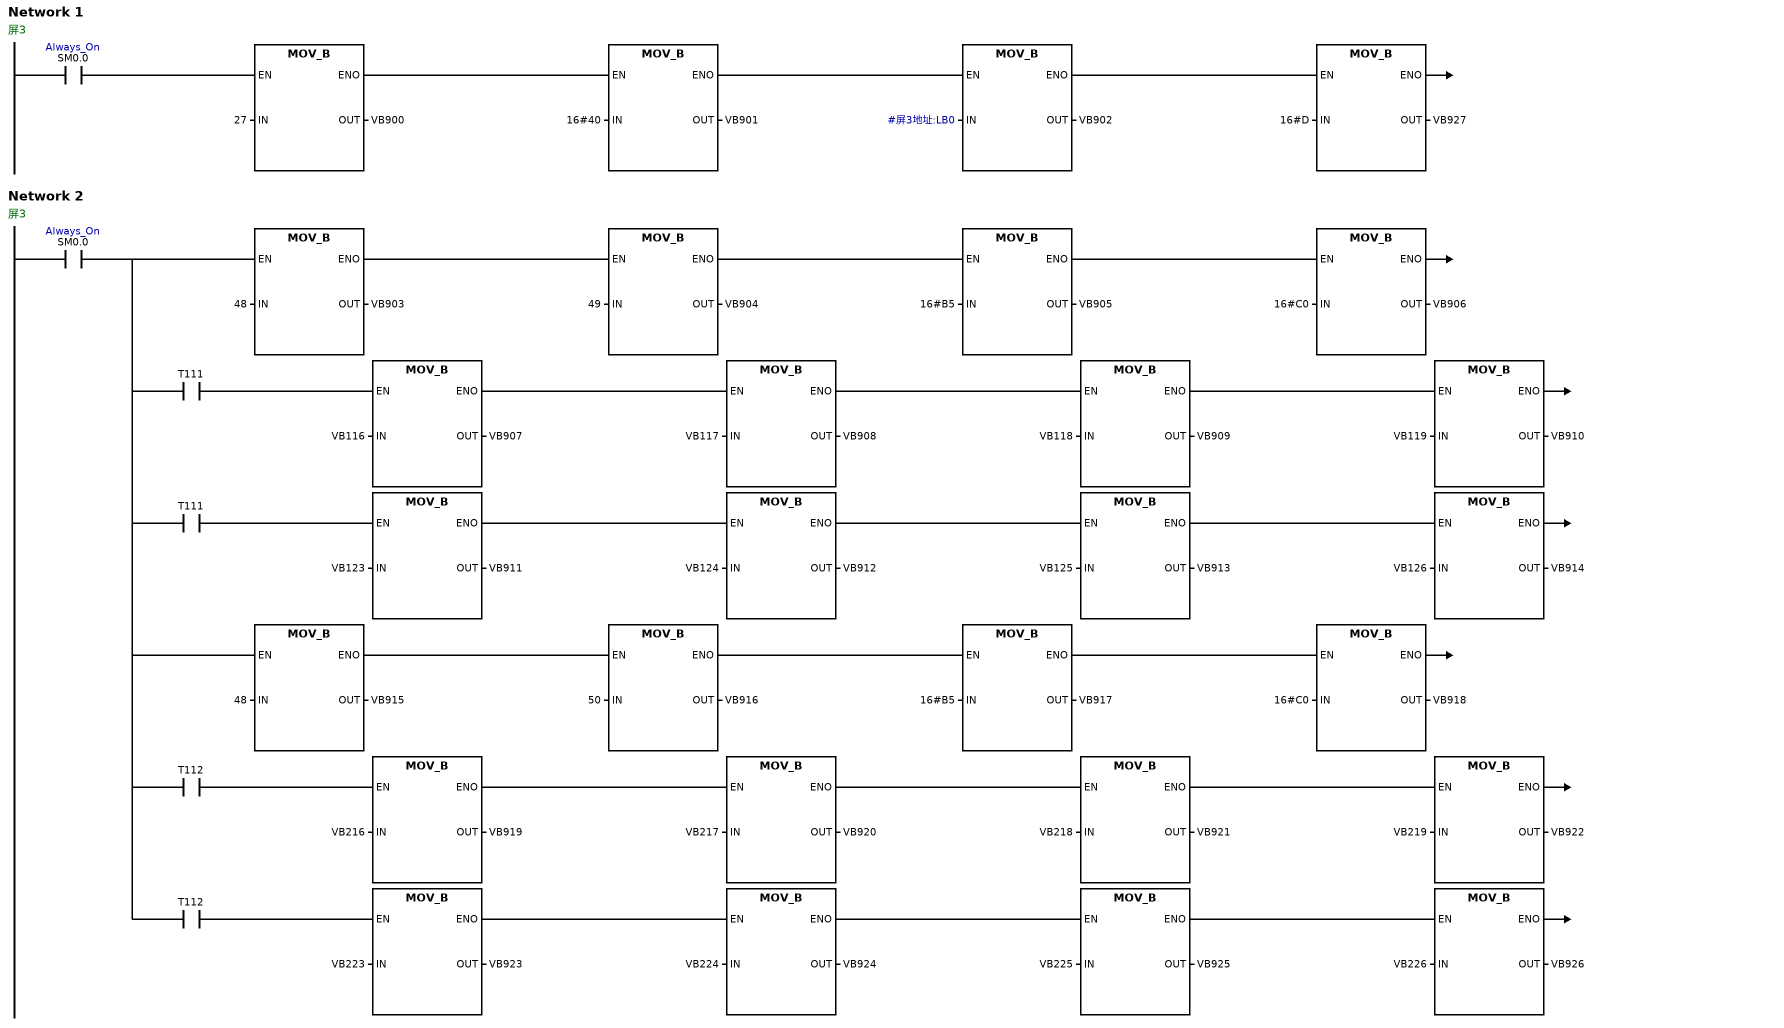
Network 1
// 屏3
LD     Always_On:SM0.0
MOVB   27, VB900
AENO
MOVB   16#40, VB901
AENO
MOVB   #屏3地址:LB0, VB902
AENO
MOVB   16#D, VB927
Network 2
// 屏3
LD     Always_On:SM0.0
LPS
MOVB   48, VB903
AENO
MOVB   49, VB904
AENO
MOVB   16#B5, VB905
AENO
MOVB   16#C0, VB906
LRD
A      T111
MOVB   VB116, VB907
AENO
MOVB   VB117, VB908
AENO
MOVB   VB118, VB909
AENO
MOVB   VB119, VB910
LRD
A      T111
MOVB   VB123, VB911
AENO
MOVB   VB124, VB912
AENO
MOVB   VB125, VB913
AENO
MOVB   VB126, VB914
LRD
MOVB   48, VB915
AENO
MOVB   50, VB916
AENO
MOVB   16#B5, VB917
AENO
MOVB   16#C0, VB918
LRD
A      T112
MOVB   VB216, VB919
AENO
MOVB   VB217, VB920
AENO
MOVB   VB218, VB921
AENO
MOVB   VB219, VB922
LPP
A      T112
MOVB   VB223, VB923
AENO
MOVB   VB224, VB924
AENO
MOVB   VB225, VB925
AENO
MOVB   VB226, VB926
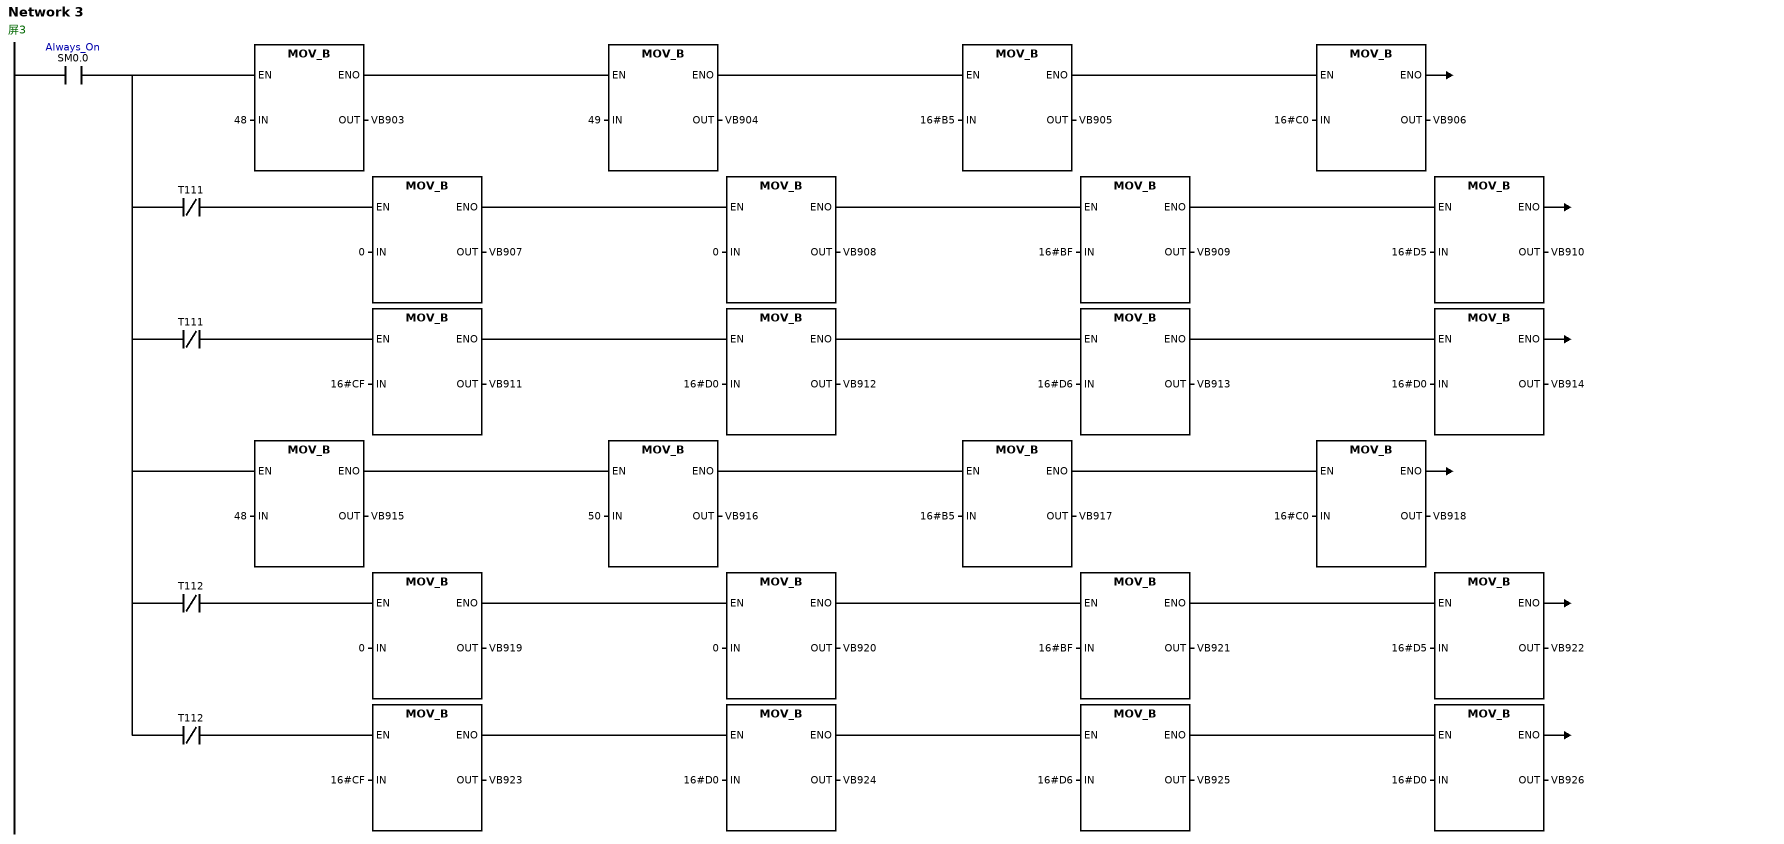
Network 3
// 屏3
LD     Always_On:SM0.0
LPS
MOVB   48, VB903
AENO
MOVB   49, VB904
AENO
MOVB   16#B5, VB905
AENO
MOVB   16#C0, VB906
LRD
AN     T111
MOVB   0, VB907
AENO
MOVB   0, VB908
AENO
MOVB   16#BF, VB909
AENO
MOVB   16#D5, VB910
LRD
AN     T111
MOVB   16#CF, VB911
AENO
MOVB   16#D0, VB912
AENO
MOVB   16#D6, VB913
AENO
MOVB   16#D0, VB914
LRD
MOVB   48, VB915
AENO
MOVB   50, VB916
AENO
MOVB   16#B5, VB917
AENO
MOVB   16#C0, VB918
LRD
AN     T112
MOVB   0, VB919
AENO
MOVB   0, VB920
AENO
MOVB   16#BF, VB921
AENO
MOVB   16#D5, VB922
LPP
AN     T112
MOVB   16#CF, VB923
AENO
MOVB   16#D0, VB924
AENO
MOVB   16#D6, VB925
AENO
MOVB   16#D0, VB926
END_SUBROUTINE_BLOCK

SUBROUTINE_BLOCK GGLED3_4:SBR32
TITLE=子程序注释
VAR_INPUT
屏3地址:BYTE;	// LB0 
END_VAR
BEGIN
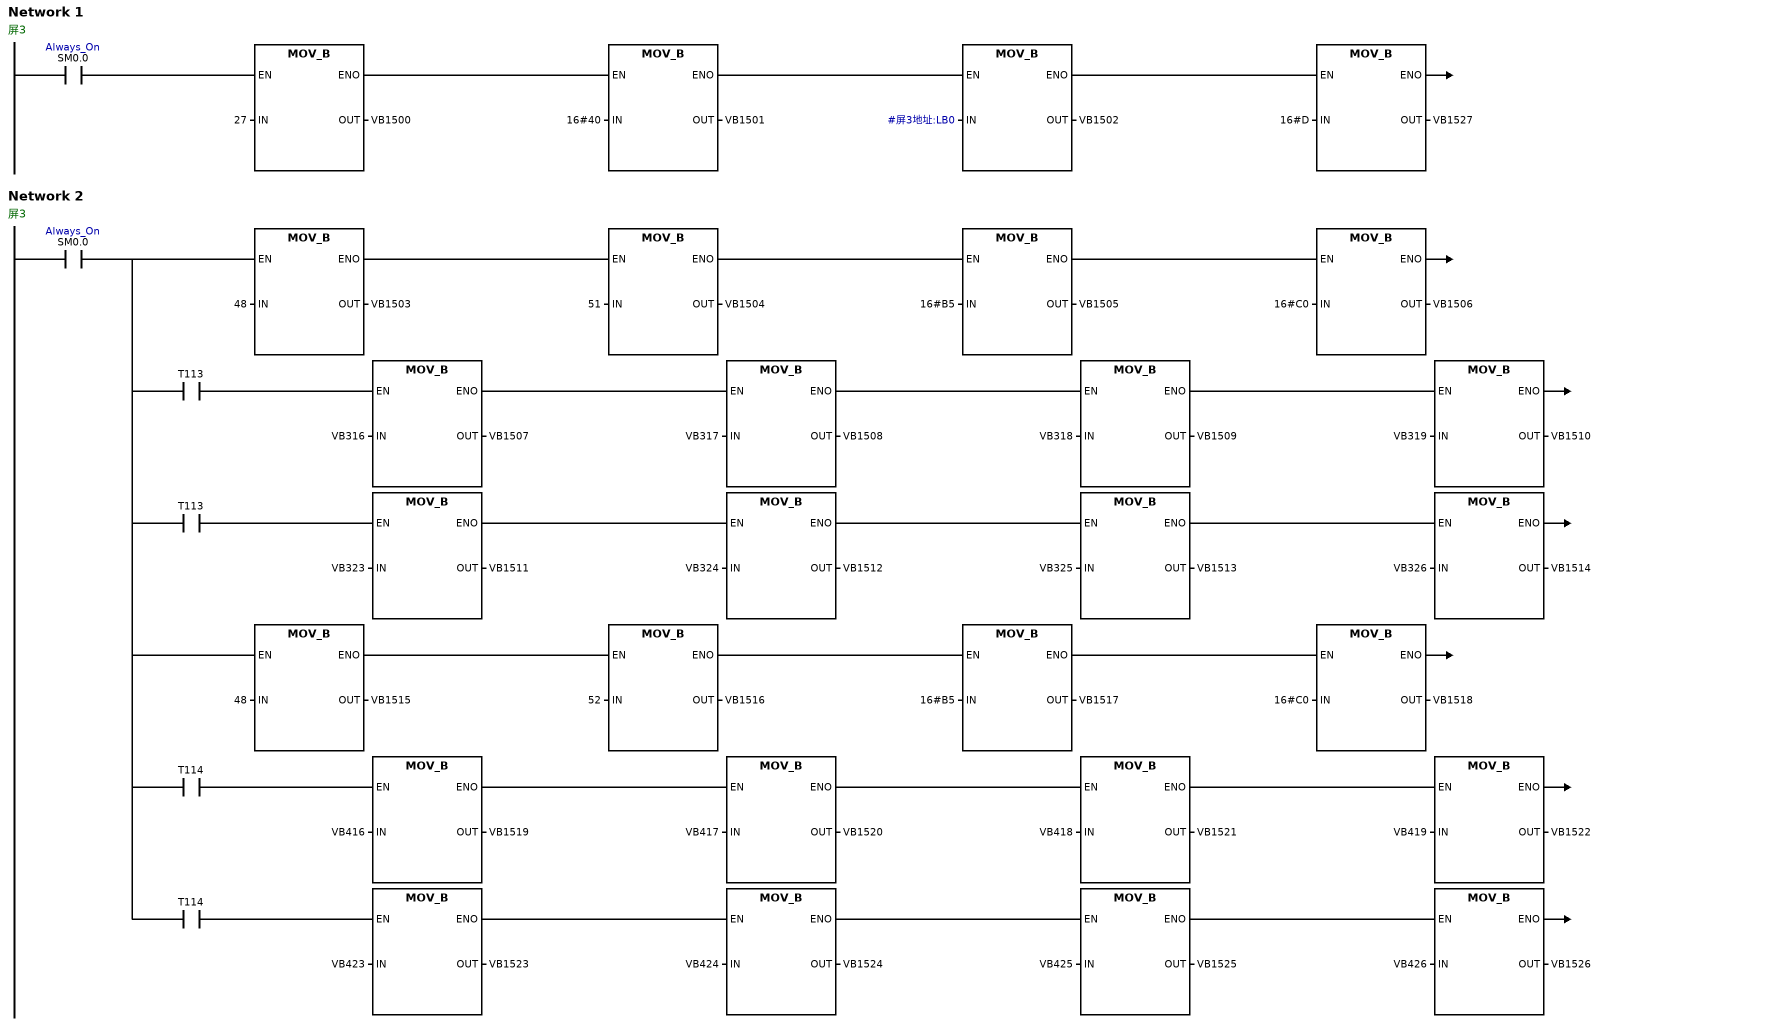
Network 1
// 屏3
LD     Always_On:SM0.0
MOVB   27, VB1500
AENO
MOVB   16#40, VB1501
AENO
MOVB   #屏3地址:LB0, VB1502
AENO
MOVB   16#D, VB1527
Network 2
// 屏3
LD     Always_On:SM0.0
LPS
MOVB   48, VB1503
AENO
MOVB   51, VB1504
AENO
MOVB   16#B5, VB1505
AENO
MOVB   16#C0, VB1506
LRD
A      T113
MOVB   VB316, VB1507
AENO
MOVB   VB317, VB1508
AENO
MOVB   VB318, VB1509
AENO
MOVB   VB319, VB1510
LRD
A      T113
MOVB   VB323, VB1511
AENO
MOVB   VB324, VB1512
AENO
MOVB   VB325, VB1513
AENO
MOVB   VB326, VB1514
LRD
MOVB   48, VB1515
AENO
MOVB   52, VB1516
AENO
MOVB   16#B5, VB1517
AENO
MOVB   16#C0, VB1518
LRD
A      T114
MOVB   VB416, VB1519
AENO
MOVB   VB417, VB1520
AENO
MOVB   VB418, VB1521
AENO
MOVB   VB419, VB1522
LPP
A      T114
MOVB   VB423, VB1523
AENO
MOVB   VB424, VB1524
AENO
MOVB   VB425, VB1525
AENO
MOVB   VB426, VB1526
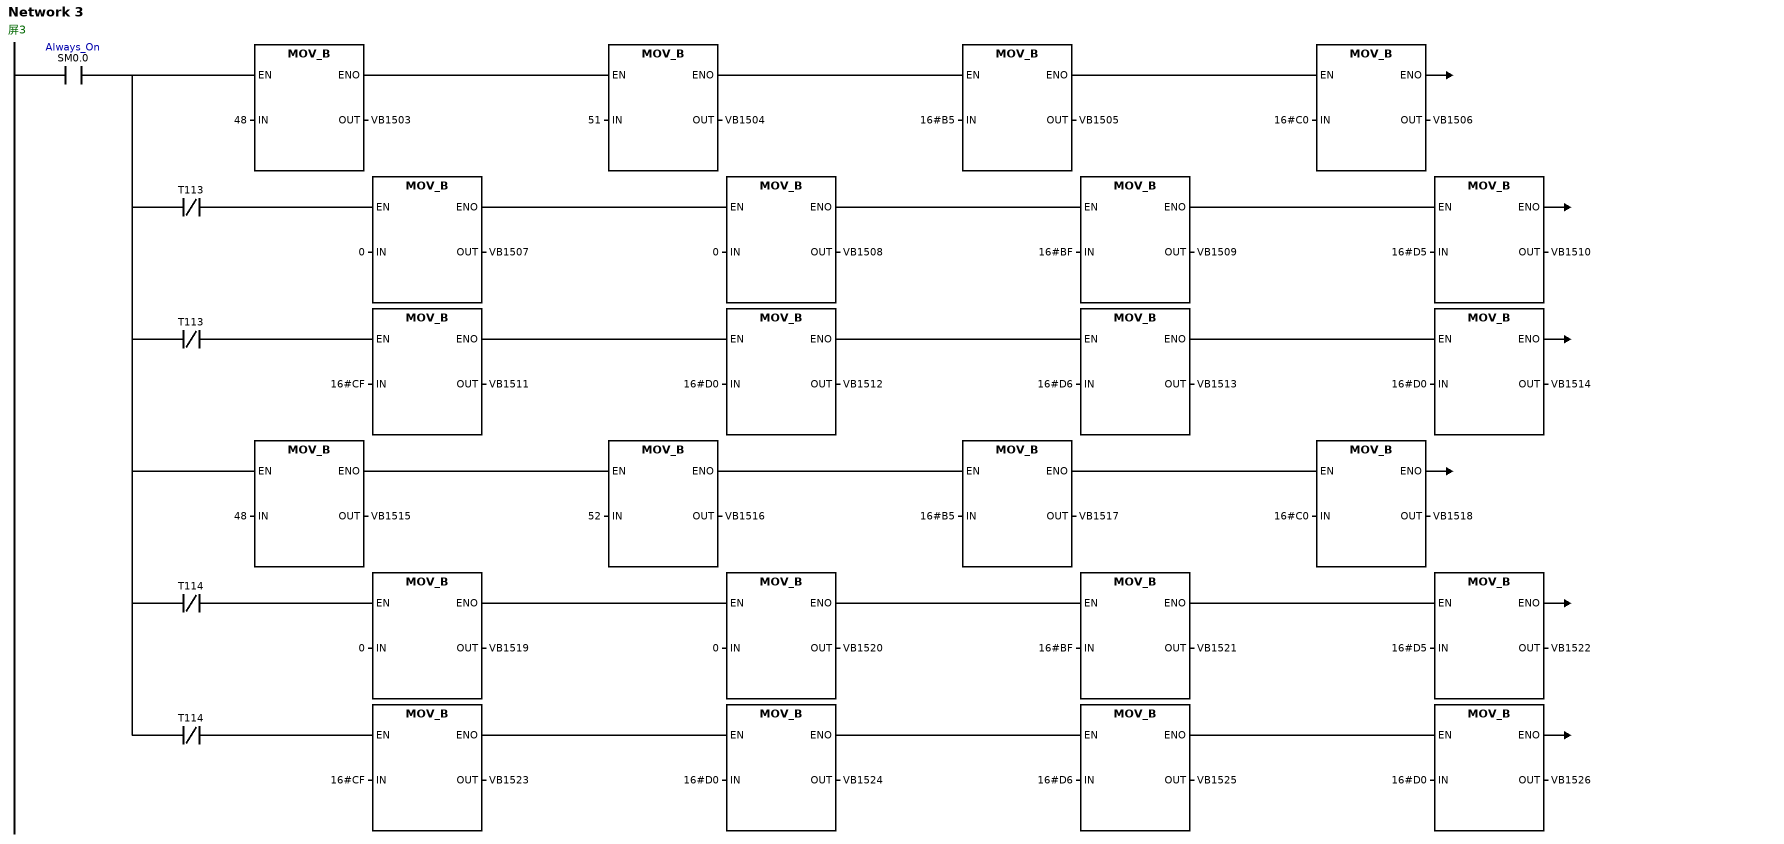
Network 3
// 屏3
LD     Always_On:SM0.0
LPS
MOVB   48, VB1503
AENO
MOVB   51, VB1504
AENO
MOVB   16#B5, VB1505
AENO
MOVB   16#C0, VB1506
LRD
AN     T113
MOVB   0, VB1507
AENO
MOVB   0, VB1508
AENO
MOVB   16#BF, VB1509
AENO
MOVB   16#D5, VB1510
LRD
AN     T113
MOVB   16#CF, VB1511
AENO
MOVB   16#D0, VB1512
AENO
MOVB   16#D6, VB1513
AENO
MOVB   16#D0, VB1514
LRD
MOVB   48, VB1515
AENO
MOVB   52, VB1516
AENO
MOVB   16#B5, VB1517
AENO
MOVB   16#C0, VB1518
LRD
AN     T114
MOVB   0, VB1519
AENO
MOVB   0, VB1520
AENO
MOVB   16#BF, VB1521
AENO
MOVB   16#D5, VB1522
LPP
AN     T114
MOVB   16#CF, VB1523
AENO
MOVB   16#D0, VB1524
AENO
MOVB   16#D6, VB1525
AENO
MOVB   16#D0, VB1526
END_SUBROUTINE_BLOCK

// SBR50: protected block, not included

// SBR51: protected block, not included

// SBR52: protected block, not included
